LIN {X 0,Y 153.521,Z 523.718,A -85,B 0,C 180,E1 -23960.081,E2 -23960.081} C_VEL
LIN {X 0,Y 151.125,Z 510.32,A -85,B 0,C 180,E1 -23962.603,E2 -23962.603} C_VEL
LIN {X 0,Y 149.17,Z 497.902,A -85,B 0,C 180,E1 -23964.528,E2 -23964.528} C_VEL
LIN {X 0,Y 149.562,Z 497.851,A -85,B 0,C 180,E1 -23971.125,E2 -23971.125} C_VEL
LIN {X 0,Y 149.777,Z 497.824,A -85,B 0,C 180,E1 -23974.27,E2 -23974.27} C_VEL
LIN {X 0,Y 149.994,Z 497.8,A -85,B 0,C 180,E1 -23977.527,E2 -23977.527} C_VEL
LIN {X 0,Y 150.1,Z 497.781,A -85,B 0,C 180,E1 -23981.482,E2 -23981.482} C_VEL
LIN {X 0,Y 150.129,Z 497.783,A -85,B 0,C 180,E1 -23985.396,E2 -23985.396} C_VEL
LIN {X 0,Y 150.159,Z 497.776,A -85,B 0,C 180,E1 -23989.06,E2 -23989.06} C_VEL
LIN {X 0,Y 150.219,Z 497.772,A -85,B 0,C 180,E1 -23992.689,E2 -23992.689} C_VEL
LIN {X 0,Y 150.222,Z 497.77,A -85,B 0,C 180,E1 -23997.365,E2 -23997.365} C_VEL
LIN {X 0,Y 150.249,Z 497.769,A -85,B 0,C 180,E1 -24002.717,E2 -24002.717} C_VEL
LIN {X 0,Y 150.355,Z 497.751,A -85,B 0,C 180,E1 -24009.207,E2 -24009.207} C_VEL
LIN {X 0,Y 150.367,Z 497.755,A -85,B 0,C 180,E1 -24013.713,E2 -24013.713} C_VEL
LIN {X 0,Y 150.616,Z 497.721,A -85,B 0,C 180,E1 -24019.242,E2 -24019.242} C_VEL
LIN {X 0,Y 150.709,Z 497.713,A -85,B 0,C 180,E1 -24021.957,E2 -24021.957} C_VEL
LIN {X 0,Y 151.222,Z 497.65,A -85,B 0,C 180,E1 -24029.999,E2 -24029.999} C_VEL
LIN {X 0,Y 150.706,Z 497.714,A -85,B 0,C 180,E1 -24038.042,E2 -24038.042} C_VEL
LIN {X 0,Y 150.581,Z 497.726,A -85,B 0,C 180,E1 -24041.437,E2 -24041.437} C_VEL
LIN {X 0,Y 150.366,Z 497.755,A -85,B 0,C 180,E1 -24046.286,E2 -24046.286} C_VEL
LIN {X 0,Y 150.354,Z 497.751,A -85,B 0,C 180,E1 -24050.792,E2 -24050.792} C_VEL
LIN {X 0,Y 150.247,Z 497.769,A -85,B 0,C 180,E1 -24057.282,E2 -24057.282} C_VEL
LIN {X 0,Y 150.221,Z 497.77,A -85,B 0,C 180,E1 -24062.634,E2 -24062.634} C_VEL
LIN {X 0,Y 150.213,Z 497.773,A -85,B 0,C 180,E1 -24067.461,E2 -24067.461} C_VEL
LIN {X 0,Y 150.155,Z 497.778,A -85,B 0,C 180,E1 -24071.505,E2 -24071.505} C_VEL
LIN {X 0,Y 150.127,Z 497.784,A -85,B 0,C 180,E1 -24075.395,E2 -24075.395} C_VEL
LIN {X 0,Y 150.151,Z 497.775,A -85,B 0,C 180,E1 -24079.057,E2 -24079.057} C_VEL
LIN {X 0,Y 150.18,Z 497.777,A -85,B 0,C 180,E1 -24082.707,E2 -24082.707} C_VEL
LIN {X 0,Y 150.216,Z 497.767,A -85,B 0,C 180,E1 -24087.367,E2 -24087.367} C_VEL
LIN {X 0,Y 150.246,Z 497.768,A -85,B 0,C 180,E1 -24092.717,E2 -24092.717} C_VEL
LIN {X 0,Y 150.352,Z 497.756,A -85,B 0,C 180,E1 -24099.207,E2 -24099.207} C_VEL
LIN {X 0,Y 150.369,Z 497.749,A -85,B 0,C 180,E1 -24103.713,E2 -24103.713} C_VEL
LIN {X 0,Y 150.689,Z 497.715,A -85,B 0,C 180,E1 -24109.247,E2 -24109.247} C_VEL
LIN {X 0,Y 150.764,Z 497.701,A -85,B 0,C 180,E1 -24111.96,E2 -24111.96} C_VEL
LIN {X 0,Y 151.219,Z 497.646,A -85,B 0,C 180,E1 -24119.999,E2 -24119.999} C_VEL
LIN {X 0,Y 150.763,Z 497.704,A -85,B 0,C 180,E1 -24128.038,E2 -24128.038} C_VEL
LIN {X 0,Y 150.635,Z 497.716,A -85,B 0,C 180,E1 -24131.546,E2 -24131.546} C_VEL
LIN {X 0,Y 150.39,Z 497.75,A -85,B 0,C 180,E1 -24136.283,E2 -24136.283} C_VEL
LIN {X 0,Y 150.352,Z 497.751,A -85,B 0,C 180,E1 -24140.793,E2 -24140.793} C_VEL
LIN {X 0,Y 150.243,Z 497.766,A -85,B 0,C 180,E1 -24147.282,E2 -24147.282} C_VEL
LIN {X 0,Y 150.217,Z 497.772,A -85,B 0,C 180,E1 -24152.634,E2 -24152.634} C_VEL
LIN {X 0,Y 150.272,Z 497.761,A -85,B 0,C 180,E1 -24157.444,E2 -24157.444} C_VEL
LIN {X 0,Y 150.66,Z 497.722,A -85,B 0,C 180,E1 -24164.404,E2 -24164.404} C_VEL
LIN {X 0,Y 150.926,Z 497.779,A -85,B 0,C 180,E1 -24167.801,E2 -24167.801} C_VEL
LIN {X 0,Y 151.492,Z 501.356,A -85,B 0,C 180,E1 -24172.909,E2 -24172.909} C_VEL
LIN {X 0,Y 150.914,Z 503.56,A -85,B 0,C 180,E1 -24176.025,E2 -24176.025} C_VEL
LIN {X 0,Y 149.311,Z 508.708,A -85,B 0,C 180,E1 -24183.421,E2 -24183.421} C_VEL
LIN {X 0,Y 149.153,Z 509.709,A -85,B 0,C 180,E1 -24184.554,E2 -24184.554} C_VEL
LIN {X 0,Y 149.244,Z 521.963,A -85,B 0,C 180,E1 -24186.221,E2 -24186.221} C_VEL
LIN {X 0,Y 150.04,Z 534.433,A -85,B 0,C 180,E1 -24188.353,E2 -24188.353} C_VEL
LIN {X 0,Y 151.472,Z 548.682,A -85,B 0,C 180,E1 -24191.399,E2 -24191.399} C_VEL
LIN {X 0,Y 152.465,Z 556.019,A -85,B 0,C 180,E1 -24193.256,E2 -24193.256} C_VEL
LIN {X 0,Y 151.39,Z 566.543,A -85,B 0,C 180,E1 -24196.579,E2 -24196.579} C_VEL
LIN {X 0,Y 150.754,Z 575.217,A -85,B 0,C 180,E1 -24199.935,E2 -24199.935} C_VEL
LIN {X 0,Y 150.469,Z 583.731,A -85,B 0,C 180,E1 -24203.968,E2 -24203.968} C_VEL
LIN {X 0,Y 150.485,Z 590.632,A -85,B 0,C 180,E1 -24207.993,E2 -24207.993} C_VEL
LIN {X 0,Y 150.437,Z 595.255,A -85,B 0,C 180,E1 -24211.339,E2 -24211.339} C_VEL
LIN {X 0,Y 149.675,Z 599.338,A -85,B 0,C 180,E1 -24215.389,E2 -24215.389} C_VEL
LIN {X 0,Y 149.531,Z 603.504,A -85,B 0,C 180,E1 -24220.837,E2 -24220.837} C_VEL
LIN {X 0,Y 150.784,Z 606.344,A -85,B 0,C 180,E1 -24226.24,E2 -24226.24} C_VEL
LIN {X 0,Y 153.651,Z 608.104,A -85,B 0,C 180,E1 -24231.465,E2 -24231.465} C_VEL
LIN {X 0,Y 158.091,Z 608.839,A -85,B 0,C 180,E1 -24236.395,E2 -24236.395} C_VEL
LIN {X 0,Y 163.869,Z 608.541,A -85,B 0,C 180,E1 -24240.975,E2 -24240.975} C_VEL
LIN {X 0,Y 171.129,Z 607.246,A -85,B 0,C 180,E1 -24245.097,E2 -24245.097} C_VEL
LIN {X 0,Y 179.626,Z 604.926,A -85,B 0,C 180,E1 -24248.757,E2 -24248.757} C_VEL
LIN {X 0,Y 189.105,Z 601.572,A -85,B 0,C 180,E1 -24251.988,E2 -24251.988} C_VEL
LIN {X 0,Y 192.623,Z 600.091,A -85,B 0,C 180,E1 -24253.138,E2 -24253.138} C_VEL
LIN {X 0,Y 193.61,Z 599.628,A -85,B 0,C 180,E1 -24253.607,E2 -24253.607} C_VEL
LIN {X 0,Y 196.664,Z 597.909,A -85,B 0,C 180,E1 -24255.621,E2 -24255.621} C_VEL
LIN {X 0,Y 197.814,Z 597.023,A -85,B 0,C 180,E1 -24257.543,E2 -24257.543} C_VEL
LIN {X 0,Y 197.818,Z 596.879,A -85,B 0,C 180,E1 -24258.253,E2 -24258.253} C_VEL
LIN {X 0,Y 195.704,Z 597.395,A -85,B 0,C 180,E1 -24259.729,E2 -24259.729} C_VEL
LIN {X 0,Y 186.845,Z 599.739,A -85,B 0,C 180,E1 -24262.461,E2 -24262.461} C_VEL
LIN {X 0,Y 182.52,Z 600.628,A -85,B 0,C 180,E1 -24263.684,E2 -24263.684} C_VEL
LIN {X 0,Y 174.385,Z 601.787,A -85,B 0,C 180,E1 -24265.473,E2 -24265.473} C_VEL
LIN {X 0,Y 166.565,Z 602.246,A -85,B 0,C 180,E1 -24267.481,E2 -24267.481} C_VEL
LIN {X 0,Y 162.816,Z 602.037,A -85,B 0,C 180,E1 -24269.048,E2 -24269.048} C_VEL
LIN {X 0,Y 156.211,Z 600.761,A -85,B 0,C 180,E1 -24273.263,E2 -24273.263} C_VEL
LIN {X 0,Y 150.578,Z 598.332,A -85,B 0,C 180,E1 -24278.076,E2 -24278.076} C_VEL
LIN {X 0,Y 146.248,Z 594.729,A -85,B 0,C 180,E1 -24283.242,E2 -24283.242} C_VEL
LIN {X 0,Y 143.432,Z 589.927,A -85,B 0,C 180,E1 -24288.698,E2 -24288.698} C_VEL
LIN {X 0,Y 142.119,Z 583.755,A -85,B 0,C 180,E1 -24294.325,E2 -24294.325} C_VEL
LIN {X 0,Y 141.676,Z 576.967,A -85,B 0,C 180,E1 -24299.29,E2 -24299.29} C_VEL
LIN {X 0,Y 141.77,Z 569.83,A -85,B 0,C 180,E1 -24303.553,E2 -24303.553} C_VEL
LIN {X 0,Y 142.26,Z 561.329,A -85,B 0,C 180,E1 -24307.791,E2 -24307.791} C_VEL
LIN {X 0,Y 143.209,Z 550.91,A -85,B 0,C 180,E1 -24312.039,E2 -24312.039} C_VEL
LIN {X 0,Y 144.511,Z 539.254,A -85,B 0,C 180,E1 -24315.877,E2 -24315.877} C_VEL
LIN {X 0,Y 146.135,Z 526.358,A -85,B 0,C 180,E1 -24319.308,E2 -24319.308} C_VEL
LIN {X 0,Y 146.371,Z 523.299,A -85,B 0,C 180,E1 -24319.997,E2 -24319.997} C_VEL
LIN {X 0,Y 144.062,Z 510.827,A -85,B 0,C 180,E1 -24322.434,E2 -24322.434} C_VEL
LIN {X 0,Y 142.132,Z 498.779,A -85,B 0,C 180,E1 -24324.368,E2 -24324.368} C_VEL
LIN {X 0,Y 142.327,Z 498.755,A -85,B 0,C 180,E1 -24329.591,E2 -24329.591} C_VEL
LIN {X 0,Y 142.661,Z 498.708,A -85,B 0,C 180,E1 -24333.123,E2 -24333.123} C_VEL
LIN {X 0,Y 142.93,Z 498.682,A -85,B 0,C 180,E1 -24338.117,E2 -24338.117} C_VEL
LIN {X 0,Y 143.026,Z 498.665,A -85,B 0,C 180,E1 -24343.468,E2 -24343.468} C_VEL
LIN {X 0,Y 143.071,Z 498.662,A -85,B 0,C 180,E1 -24347.464,E2 -24347.464} C_VEL
LIN {X 0,Y 143.11,Z 498.654,A -85,B 0,C 180,E1 -24351.791,E2 -24351.791} C_VEL
LIN {X 0,Y 143.19,Z 498.646,A -85,B 0,C 180,E1 -24357.322,E2 -24357.322} C_VEL
LIN {X 0,Y 143.195,Z 498.647,A -85,B 0,C 180,E1 -24362.062,E2 -24362.062} C_VEL
LIN {X 0,Y 143.281,Z 498.633,A -85,B 0,C 180,E1 -24368.745,E2 -24368.745} C_VEL
LIN {X 0,Y 143.306,Z 498.633,A -85,B 0,C 180,E1 -24372.887,E2 -24372.887} C_VEL
LIN {X 0,Y 143.542,Z 498.603,A -85,B 0,C 180,E1 -24378.705,E2 -24378.705} C_VEL
LIN {X 0,Y 143.631,Z 498.594,A -85,B 0,C 180,E1 -24381.558,E2 -24381.558} C_VEL
LIN {X 0,Y 144.18,Z 498.527,A -85,B 0,C 180,E1 -24389.999,E2 -24389.999} C_VEL
LIN {X 0,Y 143.628,Z 498.594,A -85,B 0,C 180,E1 -24398.441,E2 -24398.441} C_VEL
LIN {X 0,Y 143.509,Z 498.606,A -85,B 0,C 180,E1 -24401.63,E2 -24401.63} C_VEL
LIN {X 0,Y 143.305,Z 498.633,A -85,B 0,C 180,E1 -24407.112,E2 -24407.112} C_VEL
LIN {X 0,Y 143.28,Z 498.633,A -85,B 0,C 180,E1 -24411.254,E2 -24411.254} C_VEL
LIN {X 0,Y 143.193,Z 498.647,A -85,B 0,C 180,E1 -24417.937,E2 -24417.937} C_VEL
LIN {X 0,Y 143.171,Z 498.649,A -85,B 0,C 180,E1 -24423.435,E2 -24423.435} C_VEL
LIN {X 0,Y 143.076,Z 498.657,A -85,B 0,C 180,E1 -24429.684,E2 -24429.684} C_VEL
LIN {X 0,Y 143.058,Z 498.665,A -85,B 0,C 180,E1 -24433.454,E2 -24433.454} C_VEL
LIN {X 0,Y 143.066,Z 498.659,A -85,B 0,C 180,E1 -24437.464,E2 -24437.464} C_VEL
LIN {X 0,Y 143.079,Z 498.663,A -85,B 0,C 180,E1 -24441.805,E2 -24441.805} C_VEL
LIN {X 0,Y 143.183,Z 498.643,A -85,B 0,C 180,E1 -24447.321,E2 -24447.321} C_VEL
LIN {X 0,Y 143.192,Z 498.648,A -85,B 0,C 180,E1 -24452.061,E2 -24452.061} C_VEL
LIN {X 0,Y 143.278,Z 498.636,A -85,B 0,C 180,E1 -24458.744,E2 -24458.744} C_VEL
LIN {X 0,Y 143.306,Z 498.631,A -85,B 0,C 180,E1 -24462.887,E2 -24462.887} C_VEL
LIN {X 0,Y 143.603,Z 498.596,A -85,B 0,C 180,E1 -24468.71,E2 -24468.71} C_VEL
LIN {X 0,Y 143.685,Z 498.584,A -85,B 0,C 180,E1 -24471.561,E2 -24471.561} C_VEL
LIN {X 0,Y 144.178,Z 498.523,A -85,B 0,C 180,E1 -24479.999,E2 -24479.999} C_VEL
LIN {X 0,Y 143.685,Z 498.585,A -85,B 0,C 180,E1 -24488.437,E2 -24488.437} C_VEL
LIN {X 0,Y 143.571,Z 498.597,A -85,B 0,C 180,E1 -24491.757,E2 -24491.757} C_VEL
LIN {X 0,Y 143.323,Z 498.632,A -85,B 0,C 180,E1 -24497.11,E2 -24497.11} C_VEL
LIN {X 0,Y 143.277,Z 498.634,A -85,B 0,C 180,E1 -24501.255,E2 -24501.255} C_VEL
LIN {X 0,Y 143.189,Z 498.642,A -85,B 0,C 180,E1 -24507.937,E2 -24507.937} C_VEL
LIN {X 0,Y 143.169,Z 498.652,A -85,B 0,C 180,E1 -24513.436,E2 -24513.436} C_VEL
LIN {X 0,Y 143.235,Z 498.642,A -85,B 0,C 180,E1 -24519.632,E2 -24519.632} C_VEL
LIN {X 0,Y 143.47,Z 498.614,A -85,B 0,C 180,E1 -24523.298,E2 -24523.298} C_VEL
LIN {X 0,Y 143.966,Z 498.62,A -85,B 0,C 180,E1 -24528.703,E2 -24528.703} C_VEL
LIN {X 0,Y 144.404,Z 501.33,A -85,B 0,C 180,E1 -24532.773,E2 -24532.773} C_VEL
LIN {X 0,Y 143.396,Z 504.406,A -85,B 0,C 180,E1 -24537.377,E2 -24537.377} C_VEL
LIN {X 0,Y 142.08,Z 509.031,A -85,B 0,C 180,E1 -24544.452,E2 -24544.452} C_VEL
LIN {X 0,Y 142.227,Z 522.949,A -85,B 0,C 180,E1 -24546.522,E2 -24546.522} C_VEL
LIN {X 0,Y 143.214,Z 536.813,A -85,B 0,C 180,E1 -24549.131,E2 -24549.131} C_VEL
LIN {X 0,Y 144.534,Z 549.001,A -85,B 0,C 180,E1 -24551.942,E2 -24551.942} C_VEL
LIN {X 0,Y 145.421,Z 554.89,A -85,B 0,C 180,E1 -24553.506,E2 -24553.506} C_VEL
LIN {X 0,Y 144.47,Z 565.324,A -85,B 0,C 180,E1 -24556.981,E2 -24556.981} C_VEL
LIN {X 0,Y 143.853,Z 574.877,A -85,B 0,C 180,E1 -24560.864,E2 -24560.864} C_VEL
LIN {X 0,Y 143.686,Z 583.335,A -85,B 0,C 180,E1 -24565.09,E2 -24565.09} C_VEL
LIN {X 0,Y 143.719,Z 589.07,A -85,B 0,C 180,E1 -24568.6,E2 -24568.6} C_VEL
LIN {X 0,Y 143.714,Z 592.828,A -85,B 0,C 180,E1 -24571.402,E2 -24571.402} C_VEL
LIN {X 0,Y 143.198,Z 595.868,A -85,B 0,C 180,E1 -24574.222,E2 -24574.222} C_VEL
LIN {X 0,Y 142.722,Z 600.711,A -85,B 0,C 180,E1 -24579.988,E2 -24579.988} C_VEL
LIN {X 0,Y 143.292,Z 603.359,A -85,B 0,C 180,E1 -24584.196,E2 -24584.196} C_VEL
LIN {X 0,Y 145.395,Z 605.94,A -85,B 0,C 180,E1 -24589.778,E2 -24589.778} C_VEL
LIN {X 0,Y 149.33,Z 607.531,A -85,B 0,C 180,E1 -24595.061,E2 -24595.061} C_VEL
LIN {X 0,Y 154.681,Z 608.094,A -85,B 0,C 180,E1 -24599.987,E2 -24599.987} C_VEL
LIN {X 0,Y 161.446,Z 607.693,A -85,B 0,C 180,E1 -24604.466,E2 -24604.466} C_VEL
LIN {X 0,Y 169.632,Z 606.322,A -85,B 0,C 180,E1 -24608.424,E2 -24608.424} C_VEL
LIN {X 0,Y 178.912,Z 603.955,A -85,B 0,C 180,E1 -24611.898,E2 -24611.898} C_VEL
LIN {X 0,Y 183.913,Z 602.406,A -85,B 0,C 180,E1 -24613.461,E2 -24613.461} C_VEL
LIN {X 0,Y 188.351,Z 600.741,A -85,B 0,C 180,E1 -24615.15,E2 -24615.15} C_VEL
LIN {X 0,Y 190.86,Z 599.403,A -85,B 0,C 180,E1 -24617.431,E2 -24617.431} C_VEL
LIN {X 0,Y 190.34,Z 599.38,A -85,B 0,C 180,E1 -24618.347,E2 -24618.347} C_VEL
LIN {X 0,Y 180.398,Z 601.373,A -85,B 0,C 180,E1 -24621.441,E2 -24621.441} C_VEL
LIN {X 0,Y 171.242,Z 602.278,A -85,B 0,C 180,E1 -24624.93,E2 -24624.93} C_VEL
LIN {X 0,Y 162.816,Z 602.037,A -85,B 0,C 180,E1 -24629.048,E2 -24629.048} C_VEL
LIN {X 0,Y 159.227,Z 601.639,A -85,B 0,C 180,E1 -24630.708,E2 -24630.708} C_VEL
LIN {X 0,Y 152.249,Z 600.466,A -85,B 0,C 180,E1 -24633.261,E2 -24633.261} C_VEL
LIN {X 0,Y 145.778,Z 598.59,A -85,B 0,C 180,E1 -24636.045,E2 -24636.045} C_VEL
LIN {X 0,Y 143.074,Z 597.163,A -85,B 0,C 180,E1 -24638.044,E2 -24638.044} C_VEL
LIN {X 0,Y 138.628,Z 592.71,A -85,B 0,C 180,E1 -24643.81,E2 -24643.81} C_VEL
LIN {X 0,Y 136.116,Z 587.195,A -85,B 0,C 180,E1 -24649.635,E2 -24649.635} C_VEL
LIN {X 0,Y 135.22,Z 582.148,A -85,B 0,C 180,E1 -24654.034,E2 -24654.034} C_VEL
LIN {X 0,Y 134.779,Z 574.999,A -85,B 0,C 180,E1 -24659.254,E2 -24659.254} C_VEL
LIN {X 0,Y 134.894,Z 567.52,A -85,B 0,C 180,E1 -24663.735,E2 -24663.735} C_VEL
LIN {X 0,Y 135.401,Z 558.506,A -85,B 0,C 180,E1 -24668.188,E2 -24668.188} C_VEL
LIN {X 0,Y 136.447,Z 547.54,A -85,B 0,C 180,E1 -24672.646,E2 -24672.646} C_VEL
LIN {X 0,Y 137.713,Z 536.486,A -85,B 0,C 180,E1 -24676.302,E2 -24676.302} C_VEL
LIN {X 0,Y 139.214,Z 524.261,A -85,B 0,C 180,E1 -24679.54,E2 -24679.54} C_VEL
LIN {X 0,Y 138.497,Z 519.379,A -85,B 0,C 180,E1 -24680.613,E2 -24680.613} C_VEL
LIN {X 0,Y 136.138,Z 506.12,A -85,B 0,C 180,E1 -24683.145,E2 -24683.145} C_VEL
LIN {X 0,Y 135.091,Z 499.655,A -85,B 0,C 180,E1 -24684.279,E2 -24684.279} C_VEL
LIN {X 0,Y 135.394,Z 499.616,A -85,B 0,C 180,E1 -24691.271,E2 -24691.271} C_VEL
LIN {X 0,Y 135.681,Z 499.582,A -85,B 0,C 180,E1 -24694.736,E2 -24694.736} C_VEL
LIN {X 0,Y 135.927,Z 499.551,A -85,B 0,C 180,E1 -24699.143,E2 -24699.143} C_VEL
LIN {X 0,Y 135.973,Z 499.544,A -85,B 0,C 180,E1 -24703.645,E2 -24703.645} C_VEL
LIN {X 0,Y 136.035,Z 499.539,A -85,B 0,C 180,E1 -24707.807,E2 -24707.807} C_VEL
LIN {X 0,Y 136.059,Z 499.531,A -85,B 0,C 180,E1 -24711.694,E2 -24711.694} C_VEL
LIN {X 0,Y 136.094,Z 499.532,A -85,B 0,C 180,E1 -24715.717,E2 -24715.717} C_VEL
LIN {X 0,Y 136.151,Z 499.526,A -85,B 0,C 180,E1 -24722.317,E2 -24722.317} C_VEL
LIN {X 0,Y 136.248,Z 499.509,A -85,B 0,C 180,E1 -24728.833,E2 -24728.833} C_VEL
LIN {X 0,Y 136.273,Z 499.507,A -85,B 0,C 180,E1 -24735.056,E2 -24735.056} C_VEL
LIN {X 0,Y 136.449,Z 499.484,A -85,B 0,C 180,E1 -24738.138,E2 -24738.138} C_VEL
LIN {X 0,Y 136.556,Z 499.474,A -85,B 0,C 180,E1 -24741.117,E2 -24741.117} C_VEL
LIN {X 0,Y 137.137,Z 499.404,A -85,B 0,C 180,E1 -24749.999,E2 -24749.999} C_VEL
LIN {X 0,Y 136.553,Z 499.474,A -85,B 0,C 180,E1 -24758.881,E2 -24758.881} C_VEL
LIN {X 0,Y 136.444,Z 499.484,A -85,B 0,C 180,E1 -24761.889,E2 -24761.889} C_VEL
LIN {X 0,Y 136.245,Z 499.514,A -85,B 0,C 180,E1 -24768.028,E2 -24768.028} C_VEL
LIN {X 0,Y 136.201,Z 499.513,A -85,B 0,C 180,E1 -24771.748,E2 -24771.748} C_VEL
LIN {X 0,Y 136.103,Z 499.528,A -85,B 0,C 180,E1 -24778.616,E2 -24778.616} C_VEL
LIN {X 0,Y 136.081,Z 499.533,A -85,B 0,C 180,E1 -24784.617,E2 -24784.617} C_VEL
LIN {X 0,Y 136.052,Z 499.532,A -85,B 0,C 180,E1 -24789.207,E2 -24789.207} C_VEL
LIN {X 0,Y 136,Z 499.545,A -85,B 0,C 180,E1 -24793.657,E2 -24793.657} C_VEL
LIN {X 0,Y 136.006,Z 499.537,A -85,B 0,C 180,E1 -24797.795,E2 -24797.795} C_VEL
LIN {X 0,Y 136.028,Z 499.541,A -85,B 0,C 180,E1 -24801.683,E2 -24801.683} C_VEL
LIN {X 0,Y 136.056,Z 499.533,A -85,B 0,C 180,E1 -24805.738,E2 -24805.738} C_VEL
LIN {X 0,Y 136.148,Z 499.525,A -85,B 0,C 180,E1 -24812.316,E2 -24812.316} C_VEL
LIN {X 0,Y 136.245,Z 499.512,A -85,B 0,C 180,E1 -24818.832,E2 -24818.832} C_VEL
LIN {X 0,Y 136.278,Z 499.502,A -85,B 0,C 180,E1 -24825.056,E2 -24825.056} C_VEL
LIN {X 0,Y 136.501,Z 499.481,A -85,B 0,C 180,E1 -24828.114,E2 -24828.114} C_VEL
LIN {X 0,Y 136.609,Z 499.467,A -85,B 0,C 180,E1 -24831.121,E2 -24831.121} C_VEL
LIN {X 0,Y 137.135,Z 499.4,A -85,B 0,C 180,E1 -24839.999,E2 -24839.999} C_VEL
LIN {X 0,Y 136.609,Z 499.467,A -85,B 0,C 180,E1 -24848.878,E2 -24848.878} C_VEL
LIN {X 0,Y 136.493,Z 499.479,A -85,B 0,C 180,E1 -24851.958,E2 -24851.958} C_VEL
LIN {X 0,Y 136.257,Z 499.508,A -85,B 0,C 180,E1 -24858.027,E2 -24858.027} C_VEL
LIN {X 0,Y 136.198,Z 499.518,A -85,B 0,C 180,E1 -24861.75,E2 -24861.75} C_VEL
LIN {X 0,Y 136.099,Z 499.524,A -85,B 0,C 180,E1 -24868.616,E2 -24868.616} C_VEL
LIN {X 0,Y 136.088,Z 499.532,A -85,B 0,C 180,E1 -24874.616,E2 -24874.616} C_VEL
LIN {X 0,Y 136.179,Z 499.519,A -85,B 0,C 180,E1 -24879.275,E2 -24879.275} C_VEL
LIN {X 0,Y 136.637,Z 499.464,A -85,B 0,C 180,E1 -24886.062,E2 -24886.062} C_VEL
LIN {X 0,Y 136.997,Z 499.543,A -85,B 0,C 180,E1 -24889.896,E2 -24889.896} C_VEL
LIN {X 0,Y 137.229,Z 500.924,A -85,B 0,C 180,E1 -24892.081,E2 -24892.081} C_VEL
LIN {X 0,Y 136.801,Z 502.939,A -85,B 0,C 180,E1 -24895.283,E2 -24895.283} C_VEL
LIN {X 0,Y 135.342,Z 507.194,A -85,B 0,C 180,E1 -24902.138,E2 -24902.138} C_VEL
LIN {X 0,Y 135.005,Z 508.681,A -85,B 0,C 180,E1 -24904.567,E2 -24904.567} C_VEL
LIN {X 0,Y 135.085,Z 521.4,A -85,B 0,C 180,E1 -24906.527,E2 -24906.527} C_VEL
LIN {X 0,Y 136.027,Z 535.132,A -85,B 0,C 180,E1 -24909.195,E2 -24909.195} C_VEL
LIN {X 0,Y 137.384,Z 547.414,A -85,B 0,C 180,E1 -24912.126,E2 -24912.126} C_VEL
LIN {X 0,Y 138.4,Z 554.001,A -85,B 0,C 180,E1 -24913.934,E2 -24913.934} C_VEL
LIN {X 0,Y 137.59,Z 564.073,A -85,B 0,C 180,E1 -24917.429,E2 -24917.429} C_VEL
LIN {X 0,Y 137.047,Z 572.946,A -85,B 0,C 180,E1 -24921.151,E2 -24921.151} C_VEL
LIN {X 0,Y 136.934,Z 581.541,A -85,B 0,C 180,E1 -24925.585,E2 -24925.585} C_VEL
LIN {X 0,Y 137.016,Z 588.378,A -85,B 0,C 180,E1 -24930.001,E2 -24930.001} C_VEL
LIN {X 0,Y 136.852,Z 592.022,A -85,B 0,C 180,E1 -24932.944,E2 -24932.944} C_VEL
LIN {X 0,Y 136.035,Z 597.452,A -85,B 0,C 180,E1 -24938.917,E2 -24938.917} C_VEL
LIN {X 0,Y 136.631,Z 601.525,A -85,B 0,C 180,E1 -24944.904,E2 -24944.904} C_VEL
LIN {X 0,Y 138.872,Z 604.406,A -85,B 0,C 180,E1 -24950.749,E2 -24950.749} C_VEL
LIN {X 0,Y 143.002,Z 606.304,A -85,B 0,C 180,E1 -24956.253,E2 -24956.253} C_VEL
LIN {X 0,Y 148.6,Z 607.22,A -85,B 0,C 180,E1 -24961.349,E2 -24961.349} C_VEL
LIN {X 0,Y 155.663,Z 607.204,A -85,B 0,C 180,E1 -24965.941,E2 -24965.941} C_VEL
LIN {X 0,Y 164.135,Z 606.26,A -85,B 0,C 180,E1 -24969.963,E2 -24969.963} C_VEL
LIN {X 0,Y 173.706,Z 604.359,A -85,B 0,C 180,E1 -24973.457,E2 -24973.457} C_VEL
LIN {X 0,Y 178.839,Z 603.047,A -85,B 0,C 180,E1 -24975.021,E2 -24975.021} C_VEL
LIN {X 0,Y 182.913,Z 601.688,A -85,B 0,C 180,E1 -24976.89,E2 -24976.89} C_VEL
LIN {X 0,Y 180.034,Z 601.984,A -85,B 0,C 180,E1 -24978.423,E2 -24978.423} C_VEL
LIN {X 0,Y 169.911,Z 602.975,A -85,B 0,C 180,E1 -24981.804,E2 -24981.804} C_VEL
LIN {X 0,Y 161.223,Z 602.863,A -85,B 0,C 180,E1 -24985.48,E2 -24985.48} C_VEL
LIN {X 0,Y 153.324,Z 601.682,A -85,B 0,C 180,E1 -24989.721,E2 -24989.721} C_VEL
LIN {X 0,Y 146.749,Z 599.415,A -85,B 0,C 180,E1 -24994.468,E2 -24994.468} C_VEL
LIN {X 0,Y 143.074,Z 597.163,A -85,B 0,C 180,E1 -24998.044,E2 -24998.044} C_VEL
LIN {X 0,Y 140.599,Z 595.583,A -85,B 0,C 180,E1 -25000.104,E2 -25000.104} C_VEL
LIN {X 0,Y 135.387,Z 592.295,A -85,B 0,C 180,E1 -25003.322,E2 -25003.322} C_VEL
LIN {X 0,Y 130.782,Z 588.321,A -85,B 0,C 180,E1 -25006.709,E2 -25006.709} C_VEL
LIN {X 0,Y 129.343,Z 585.771,A -85,B 0,C 180,E1 -25008.979,E2 -25008.979} C_VEL
LIN {X 0,Y 128.353,Z 580.408,A -85,B 0,C 180,E1 -25013.714,E2 -25013.714} C_VEL
LIN {X 0,Y 127.958,Z 572.813,A -85,B 0,C 180,E1 -25019.214,E2 -25019.214} C_VEL
LIN {X 0,Y 128.057,Z 564.956,A -85,B 0,C 180,E1 -25023.934,E2 -25023.934} C_VEL
LIN {X 0,Y 128.537,Z 556.37,A -85,B 0,C 180,E1 -25028.219,E2 -25028.219} C_VEL
LIN {X 0,Y 129.525,Z 545.913,A -85,B 0,C 180,E1 -25032.536,E2 -25032.536} C_VEL
LIN {X 0,Y 130.95,Z 533.271,A -85,B 0,C 180,E1 -25036.767,E2 -25036.767} C_VEL
LIN {X 0,Y 132.118,Z 523.607,A -85,B 0,C 180,E1 -25039.42,E2 -25039.42} C_VEL
LIN {X 0,Y 129.791,Z 511.029,A -85,B 0,C 180,E1 -25042.1,E2 -25042.1} C_VEL
LIN {X 0,Y 128.1,Z 500.525,A -85,B 0,C 180,E1 -25043.974,E2 -25043.974} C_VEL
LIN {X 0,Y 128.179,Z 500.518,A -85,B 0,C 180,E1 -25049.57,E2 -25049.57} C_VEL
LIN {X 0,Y 128.634,Z 500.46,A -85,B 0,C 180,E1 -25054.96,E2 -25054.96} C_VEL
LIN {X 0,Y 128.855,Z 500.428,A -85,B 0,C 180,E1 -25060.883,E2 -25060.883} C_VEL
LIN {X 0,Y 128.919,Z 500.425,A -85,B 0,C 180,E1 -25065.13,E2 -25065.13} C_VEL
LIN {X 0,Y 128.961,Z 500.416,A -85,B 0,C 180,E1 -25069.728,E2 -25069.728} C_VEL
LIN {X 0,Y 128.996,Z 500.416,A -85,B 0,C 180,E1 -25074.811,E2 -25074.811} C_VEL
LIN {X 0,Y 129.037,Z 500.408,A -85,B 0,C 180,E1 -25080.646,E2 -25080.646} C_VEL
LIN {X 0,Y 129.112,Z 500.396,A -85,B 0,C 180,E1 -25087.602,E2 -25087.602} C_VEL
LIN {X 0,Y 129.158,Z 500.395,A -85,B 0,C 180,E1 -25090.944,E2 -25090.944} C_VEL
LIN {X 0,Y 129.37,Z 500.364,A -85,B 0,C 180,E1 -25097.922,E2 -25097.922} C_VEL
LIN {X 0,Y 129.481,Z 500.356,A -85,B 0,C 180,E1 -25100.628,E2 -25100.628} C_VEL
LIN {X 0,Y 130.092,Z 500.281,A -85,B 0,C 180,E1 -25109.999,E2 -25109.999} C_VEL
LIN {X 0,Y 129.479,Z 500.356,A -85,B 0,C 180,E1 -25119.371,E2 -25119.371} C_VEL
LIN {X 0,Y 129.347,Z 500.366,A -85,B 0,C 180,E1 -25122.552,E2 -25122.552} C_VEL
LIN {X 0,Y 129.157,Z 500.395,A -85,B 0,C 180,E1 -25129.055,E2 -25129.055} C_VEL
LIN {X 0,Y 129.111,Z 500.396,A -85,B 0,C 180,E1 -25132.397,E2 -25132.397} C_VEL
LIN {X 0,Y 129.038,Z 500.408,A -85,B 0,C 180,E1 -25139.372,E2 -25139.372} C_VEL
LIN {X 0,Y 128.994,Z 500.416,A -85,B 0,C 180,E1 -25145.188,E2 -25145.188} C_VEL
LIN {X 0,Y 128.952,Z 500.418,A -85,B 0,C 180,E1 -25150.844,E2 -25150.844} C_VEL
LIN {X 0,Y 128.923,Z 500.425,A -85,B 0,C 180,E1 -25155.126,E2 -25155.126} C_VEL
LIN {X 0,Y 128.943,Z 500.419,A -85,B 0,C 180,E1 -25159.734,E2 -25159.734} C_VEL
LIN {X 0,Y 128.96,Z 500.419,A -85,B 0,C 180,E1 -25164.831,E2 -25164.831} C_VEL
LIN {X 0,Y 129.052,Z 500.409,A -85,B 0,C 180,E1 -25170.65,E2 -25170.65} C_VEL
LIN {X 0,Y 129.108,Z 500.4,A -85,B 0,C 180,E1 -25177.727,E2 -25177.727} C_VEL
LIN {X 0,Y 129.156,Z 500.396,A -85,B 0,C 180,E1 -25180.943,E2 -25180.943} C_VEL
LIN {X 0,Y 129.418,Z 500.365,A -85,B 0,C 180,E1 -25187.815,E2 -25187.815} C_VEL
LIN {X 0,Y 129.531,Z 500.348,A -85,B 0,C 180,E1 -25190.631,E2 -25190.631} C_VEL
LIN {X 0,Y 130.09,Z 500.277,A -85,B 0,C 180,E1 -25199.999,E2 -25199.999} C_VEL
LIN {X 0,Y 129.531,Z 500.346,A -85,B 0,C 180,E1 -25209.367,E2 -25209.367} C_VEL
LIN {X 0,Y 129.395,Z 500.363,A -85,B 0,C 180,E1 -25212.547,E2 -25212.547} C_VEL
LIN {X 0,Y 129.163,Z 500.39,A -85,B 0,C 180,E1 -25219.054,E2 -25219.054} C_VEL
LIN {X 0,Y 129.108,Z 500.401,A -85,B 0,C 180,E1 -25222.398,E2 -25222.398} C_VEL
LIN {X 0,Y 129.035,Z 500.406,A -85,B 0,C 180,E1 -25229.373,E2 -25229.373} C_VEL
LIN {X 0,Y 129.036,Z 500.409,A -85,B 0,C 180,E1 -25235.217,E2 -25235.217} C_VEL
LIN {X 0,Y 129.174,Z 500.393,A -85,B 0,C 180,E1 -25240.759,E2 -25240.759} C_VEL
LIN {X 0,Y 129.485,Z 500.357,A -85,B 0,C 180,E1 -25245.123,E2 -25245.123} C_VEL
LIN {X 0,Y 130.011,Z 500.292,A -85,B 0,C 180,E1 -25250.943,E2 -25250.943} C_VEL
LIN {X 0,Y 129.902,Z 502.235,A -85,B 0,C 180,E1 -25254.246,E2 -25254.246} C_VEL
LIN {X 0,Y 128.391,Z 506.267,A -85,B 0,C 180,E1 -25261.142,E2 -25261.142} C_VEL
LIN {X 0,Y 127.932,Z 508.442,A -85,B 0,C 180,E1 -25264.694,E2 -25264.694} C_VEL
LIN {X 0,Y 128.014,Z 521.116,A -85,B 0,C 180,E1 -25266.76,E2 -25266.76} C_VEL
LIN {X 0,Y 128.876,Z 533.61,A -85,B 0,C 180,E1 -25269.301,E2 -25269.301} C_VEL
LIN {X 0,Y 130.453,Z 547.426,A -85,B 0,C 180,E1 -25272.766,E2 -25272.766} C_VEL
LIN {X 0,Y 131.45,Z 553.398,A -85,B 0,C 180,E1 -25274.496,E2 -25274.496} C_VEL
LIN {X 0,Y 130.632,Z 563.777,A -85,B 0,C 180,E1 -25278.361,E2 -25278.361} C_VEL
LIN {X 0,Y 130.251,Z 572.382,A -85,B 0,C 180,E1 -25282.248,E2 -25282.248} C_VEL
LIN {X 0,Y 130.285,Z 580.925,A -85,B 0,C 180,E1 -25286.908,E2 -25286.908} C_VEL
LIN {X 0,Y 130.345,Z 586.633,A -85,B 0,C 180,E1 -25290.773,E2 -25290.773} C_VEL
LIN {X 0,Y 130.225,Z 589.418,A -85,B 0,C 180,E1 -25293.094,E2 -25293.094} C_VEL
LIN {X 0,Y 129.383,Z 595.19,A -85,B 0,C 180,E1 -25299.379,E2 -25299.379} C_VEL
LIN {X 0,Y 130.032,Z 599.519,A -85,B 0,C 180,E1 -25305.679,E2 -25305.679} C_VEL
LIN {X 0,Y 132.441,Z 602.726,A -85,B 0,C 180,E1 -25311.806,E2 -25311.806} C_VEL
LIN {X 0,Y 136.765,Z 604.943,A -85,B 0,C 180,E1 -25317.548,E2 -25317.548} C_VEL
LIN {X 0,Y 144.864,Z 606.402,A -85,B 0,C 180,E1 -25324.438,E2 -25324.438} C_VEL
LIN {X 0,Y 154.247,Z 606.397,A -85,B 0,C 180,E1 -25329.635,E2 -25329.635} C_VEL
LIN {X 0,Y 163.577,Z 605.41,A -85,B 0,C 180,E1 -25333.428,E2 -25333.428} C_VEL
LIN {X 0,Y 173.822,Z 603.497,A -85,B 0,C 180,E1 -25336.701,E2 -25336.701} C_VEL
LIN {X 0,Y 169.652,Z 603.667,A -85,B 0,C 180,E1 -25338.486,E2 -25338.486} C_VEL
LIN {X 0,Y 159.905,Z 603.639,A -85,B 0,C 180,E1 -25342.026,E2 -25342.026} C_VEL
LIN {X 0,Y 151.168,Z 602.556,A -85,B 0,C 180,E1 -25346.09,E2 -25346.09} C_VEL
LIN {X 0,Y 143.713,Z 600.412,A -85,B 0,C 180,E1 -25350.724,E2 -25350.724} C_VEL
LIN {X 0,Y 137.574,Z 597.216,A -85,B 0,C 180,E1 -25355.878,E2 -25355.878} C_VEL
LIN {X 0,Y 132.852,Z 592.884,A -85,B 0,C 180,E1 -25361.494,E2 -25361.494} C_VEL
LIN {X 0,Y 129.78,Z 587.323,A -85,B 0,C 180,E1 -25367.491,E2 -25367.491} C_VEL
LIN {X 0,Y 129.343,Z 585.771,A -85,B 0,C 180,E1 -25368.979,E2 -25368.979} C_VEL
LIN {X 0,Y 128.156,Z 583.114,A -85,B 0,C 180,E1 -25371.24,E2 -25371.24} C_VEL
LIN {X 0,Y 124.877,Z 577.95,A -85,B 0,C 180,E1 -25374.747,E2 -25374.747} C_VEL
LIN {X 0,Y 122.325,Z 573.283,A -85,B 0,C 180,E1 -25377.55,E2 -25377.55} C_VEL
LIN {X 0,Y 121.246,Z 569.623,A -85,B 0,C 180,E1 -25379.742,E2 -25379.742} C_VEL
LIN {X 0,Y 121.151,Z 568.402,A -85,B 0,C 180,E1 -25380.497,E2 -25380.497} C_VEL
LIN {X 0,Y 121.469,Z 559.01,A -85,B 0,C 180,E1 -25385.812,E2 -25385.812} C_VEL
LIN {X 0,Y 122.336,Z 547.222,A -85,B 0,C 180,E1 -25391.234,E2 -25391.234} C_VEL
LIN {X 0,Y 123.661,Z 534.968,A -85,B 0,C 180,E1 -25395.662,E2 -25395.662} C_VEL
LIN {X 0,Y 124.996,Z 524.135,A -85,B 0,C 180,E1 -25398.863,E2 -25398.863} C_VEL
LIN {X 0,Y 124.043,Z 518.204,A -85,B 0,C 180,E1 -25400.284,E2 -25400.284} C_VEL
LIN {X 0,Y 121.36,Z 503.25,A -85,B 0,C 180,E1 -25403.299,E2 -25403.299} C_VEL
LIN {X 0,Y 121.077,Z 501.4,A -85,B 0,C 180,E1 -25403.689,E2 -25403.689} C_VEL
LIN {X 0,Y 121.226,Z 501.381,A -85,B 0,C 180,E1 -25411.452,E2 -25411.452} C_VEL
LIN {X 0,Y 121.621,Z 501.334,A -85,B 0,C 180,E1 -25416,E2 -25416} C_VEL
LIN {X 0,Y 121.796,Z 501.306,A -85,B 0,C 180,E1 -25421.396,E2 -25421.396} C_VEL
LIN {X 0,Y 121.847,Z 501.308,A -85,B 0,C 180,E1 -25426.199,E2 -25426.199} C_VEL
LIN {X 0,Y 121.877,Z 501.297,A -85,B 0,C 180,E1 -25430.63,E2 -25430.63} C_VEL
LIN {X 0,Y 121.949,Z 501.294,A -85,B 0,C 180,E1 -25434.808,E2 -25434.808} C_VEL
LIN {X 0,Y 121.946,Z 501.287,A -85,B 0,C 180,E1 -25439.826,E2 -25439.826} C_VEL
LIN {X 0,Y 121.987,Z 501.286,A -85,B 0,C 180,E1 -25446.215,E2 -25446.215} C_VEL
LIN {X 0,Y 122.049,Z 501.278,A -85,B 0,C 180,E1 -25449.787,E2 -25449.787} C_VEL
LIN {X 0,Y 122.243,Z 501.25,A -85,B 0,C 180,E1 -25456.704,E2 -25456.704} C_VEL
LIN {X 0,Y 122.411,Z 501.237,A -85,B 0,C 180,E1 -25460.081,E2 -25460.081} C_VEL
LIN {X 0,Y 122.603,Z 501.209,A -85,B 0,C 180,E1 -25466.713,E2 -25466.713} C_VEL
LIN {X 0,Y 123.045,Z 501.159,A -85,B 0,C 180,E1 -25469.999,E2 -25469.999} C_VEL
LIN {X 0,Y 122.426,Z 501.233,A -85,B 0,C 180,E1 -25476.592,E2 -25476.592} C_VEL
LIN {X 0,Y 122.321,Z 501.241,A -85,B 0,C 180,E1 -25482.375,E2 -25482.375} C_VEL
LIN {X 0,Y 122.112,Z 501.273,A -85,B 0,C 180,E1 -25486.724,E2 -25486.724} C_VEL
LIN {X 0,Y 122.026,Z 501.279,A -85,B 0,C 180,E1 -25492.85,E2 -25492.85} C_VEL
LIN {X 0,Y 121.952,Z 501.294,A -85,B 0,C 180,E1 -25497.453,E2 -25497.453} C_VEL
LIN {X 0,Y 121.914,Z 501.291,A -85,B 0,C 180,E1 -25501.253,E2 -25501.253} C_VEL
LIN {X 0,Y 121.914,Z 501.298,A -85,B 0,C 180,E1 -25506.188,E2 -25506.188} C_VEL
LIN {X 0,Y 121.886,Z 501.299,A -85,B 0,C 180,E1 -25511.444,E2 -25511.444} C_VEL
LIN {X 0,Y 121.873,Z 501.297,A -85,B 0,C 180,E1 -25518.56,E2 -25518.56} C_VEL
LIN {X 0,Y 121.912,Z 501.297,A -85,B 0,C 180,E1 -25524.795,E2 -25524.795} C_VEL
LIN {X 0,Y 121.94,Z 501.295,A -85,B 0,C 180,E1 -25529.827,E2 -25529.827} C_VEL
LIN {X 0,Y 121.984,Z 501.284,A -85,B 0,C 180,E1 -25536.214,E2 -25536.214} C_VEL
LIN {X 0,Y 122.047,Z 501.283,A -85,B 0,C 180,E1 -25539.786,E2 -25539.786} C_VEL
LIN {X 0,Y 122.365,Z 501.242,A -85,B 0,C 180,E1 -25547.521,E2 -25547.521} C_VEL
LIN {X 0,Y 122.457,Z 501.23,A -85,B 0,C 180,E1 -25550.085,E2 -25550.085} C_VEL
LIN {X 0,Y 122.611,Z 501.211,A -85,B 0,C 180,E1 -25556.713,E2 -25556.713} C_VEL
LIN {X 0,Y 123.044,Z 501.155,A -85,B 0,C 180,E1 -25559.999,E2 -25559.999} C_VEL
LIN {X 0,Y 122.456,Z 501.231,A -85,B 0,C 180,E1 -25566.59,E2 -25566.59} C_VEL
LIN {X 0,Y 122.457,Z 501.225,A -85,B 0,C 180,E1 -25569.914,E2 -25569.914} C_VEL
LIN {X 0,Y 122.265,Z 501.253,A -85,B 0,C 180,E1 -25573.292,E2 -25573.292} C_VEL
LIN {X 0,Y 122.051,Z 501.275,A -85,B 0,C 180,E1 -25580.211,E2 -25580.211} C_VEL
LIN {X 0,Y 121.983,Z 501.29,A -85,B 0,C 180,E1 -25583.784,E2 -25583.784} C_VEL
LIN {X 0,Y 121.941,Z 501.292,A -85,B 0,C 180,E1 -25590.174,E2 -25590.174} C_VEL
LIN {X 0,Y 122.006,Z 501.282,A -85,B 0,C 180,E1 -25596.25,E2 -25596.25} C_VEL
LIN {X 0,Y 122.287,Z 501.253,A -85,B 0,C 180,E1 -25603.602,E2 -25603.602} C_VEL
LIN {X 0,Y 122.67,Z 501.204,A -85,B 0,C 180,E1 -25608.141,E2 -25608.141} C_VEL
LIN {X 0,Y 122.951,Z 501.183,A -85,B 0,C 180,E1 -25612.546,E2 -25612.546} C_VEL
LIN {X 0,Y 122.158,Z 503.59,A -85,B 0,C 180,E1 -25616.87,E2 -25616.87} C_VEL
LIN {X 0,Y 120.865,Z 507.874,A -85,B 0,C 180,E1 -25624.837,E2 -25624.837} C_VEL
LIN {X 0,Y 121.011,Z 521.527,A -85,B 0,C 180,E1 -25627.238,E2 -25627.238} C_VEL
LIN {X 0,Y 122.033,Z 534.973,A -85,B 0,C 180,E1 -25630.225,E2 -25630.225} C_VEL
LIN {X 0,Y 123.551,Z 547.07,A -85,B 0,C 180,E1 -25633.477,E2 -25633.477} C_VEL
LIN {X 0,Y 124.53,Z 552.629,A -85,B 0,C 180,E1 -25635.171,E2 -25635.171} C_VEL
LIN {X 0,Y 123.792,Z 563.229,A -85,B 0,C 180,E1 -25639.368,E2 -25639.368} C_VEL
LIN {X 0,Y 123.477,Z 571.774,A -85,B 0,C 180,E1 -25643.464,E2 -25643.464} C_VEL
LIN {X 0,Y 123.626,Z 578.927,A -85,B 0,C 180,E1 -25647.557,E2 -25647.557} C_VEL
LIN {X 0,Y 123.762,Z 584.693,A -85,B 0,C 180,E1 -25651.628,E2 -25651.628} C_VEL
LIN {X 0,Y 123.373,Z 588.325,A -85,B 0,C 180,E1 -25654.903,E2 -25654.903} C_VEL
LIN {X 0,Y 122.815,Z 592.737,A -85,B 0,C 180,E1 -25659.886,E2 -25659.886} C_VEL
LIN {X 0,Y 123.511,Z 597.358,A -85,B 0,C 180,E1 -25666.53,E2 -25666.53} C_VEL
LIN {X 0,Y 126.111,Z 600.853,A -85,B 0,C 180,E1 -25672.962,E2 -25672.962} C_VEL
LIN {X 0,Y 130.646,Z 603.401,A -85,B 0,C 180,E1 -25678.957,E2 -25678.957} C_VEL
LIN {X 0,Y 139.148,Z 605.303,A -85,B 0,C 180,E1 -25686.088,E2 -25686.088} C_VEL
LIN {X 0,Y 148.884,Z 605.761,A -85,B 0,C 180,E1 -25691.367,E2 -25691.367} C_VEL
LIN {X 0,Y 158.509,Z 605.198,A -85,B 0,C 180,E1 -25695.188,E2 -25695.188} C_VEL
LIN {X 0,Y 163.707,Z 604.581,A -85,B 0,C 180,E1 -25696.872,E2 -25696.872} C_VEL
LIN {X 0,Y 159.307,Z 604.417,A -85,B 0,C 180,E1 -25698.568,E2 -25698.568} C_VEL
LIN {X 0,Y 149.755,Z 603.407,A -85,B 0,C 180,E1 -25702.405,E2 -25702.405} C_VEL
LIN {X 0,Y 141.269,Z 601.366,A -85,B 0,C 180,E1 -25706.823,E2 -25706.823} C_VEL
LIN {X 0,Y 134.136,Z 598.291,A -85,B 0,C 180,E1 -25711.866,E2 -25711.866} C_VEL
LIN {X 0,Y 128.547,Z 594.175,A -85,B 0,C 180,E1 -25717.499,E2 -25717.499} C_VEL
LIN {X 0,Y 123.868,Z 587.815,A -85,B 0,C 180,E1 -25724.699,E2 -25724.699} C_VEL
LIN {X 0,Y 121.874,Z 580.389,A -85,B 0,C 180,E1 -25731.712,E2 -25731.712} C_VEL
LIN {X 0,Y 121.151,Z 572.922,A -85,B 0,C 180,E1 -25737.507,E2 -25737.507} C_VEL
LIN {X 0,Y 121.151,Z 568.402,A -85,B 0,C 180,E1 -25740.497,E2 -25740.497} C_VEL
LIN {X 0,Y 120.523,Z 564.621,A -85,B 0,C 180,E1 -25742.624,E2 -25742.624} C_VEL
LIN {X 0,Y 117.987,Z 557.698,A -85,B 0,C 180,E1 -25745.812,E2 -25745.812} C_VEL
LIN {X 0,Y 115.674,Z 550.297,A -85,B 0,C 180,E1 -25748.91,E2 -25748.91} C_VEL
LIN {X 0,Y 115.466,Z 545.717,A -85,B 0,C 180,E1 -25750.819,E2 -25750.819} C_VEL
LIN {X 0,Y 116.824,Z 532.779,A -85,B 0,C 180,E1 -25755.729,E2 -25755.729} C_VEL
LIN {X 0,Y 117.886,Z 523.033,A -85,B 0,C 180,E1 -25758.69,E2 -25758.69} C_VEL
LIN {X 0,Y 115.274,Z 509.185,A -85,B 0,C 180,E1 -25761.88,E2 -25761.88} C_VEL
LIN {X 0,Y 114.079,Z 502.272,A -85,B 0,C 180,E1 -25763.273,E2 -25763.273} C_VEL
LIN {X 0,Y 114.133,Z 502.266,A -85,B 0,C 180,E1 -25770.447,E2 -25770.447} C_VEL
LIN {X 0,Y 114.588,Z 502.211,A -85,B 0,C 180,E1 -25777.123,E2 -25777.123} C_VEL
LIN {X 0,Y 114.73,Z 502.188,A -85,B 0,C 180,E1 -25782.685,E2 -25782.685} C_VEL
LIN {X 0,Y 114.804,Z 502.184,A -85,B 0,C 180,E1 -25787.669,E2 -25787.669} C_VEL
LIN {X 0,Y 114.816,Z 502.182,A -85,B 0,C 180,E1 -25792.727,E2 -25792.727} C_VEL
LIN {X 0,Y 114.873,Z 502.168,A -85,B 0,C 180,E1 -25798.932,E2 -25798.932} C_VEL
LIN {X 0,Y 114.951,Z 502.161,A -85,B 0,C 180,E1 -25806.507,E2 -25806.507} C_VEL
LIN {X 0,Y 115.015,Z 502.159,A -85,B 0,C 180,E1 -25812.209,E2 -25812.209} C_VEL
LIN {X 0,Y 115.256,Z 502.121,A -85,B 0,C 180,E1 -25817.333,E2 -25817.333} C_VEL
LIN {X 0,Y 115.37,Z 502.112,A -85,B 0,C 180,E1 -25823.001,E2 -25823.001} C_VEL
LIN {X 0,Y 115.996,Z 502.037,A -85,B 0,C 180,E1 -25829.999,E2 -25829.999} C_VEL
LIN {X 0,Y 115.367,Z 502.112,A -85,B 0,C 180,E1 -25836.997,E2 -25836.997} C_VEL
LIN {X 0,Y 115.255,Z 502.121,A -85,B 0,C 180,E1 -25842.665,E2 -25842.665} C_VEL
LIN {X 0,Y 115.014,Z 502.159,A -85,B 0,C 180,E1 -25847.789,E2 -25847.789} C_VEL
LIN {X 0,Y 114.949,Z 502.162,A -85,B 0,C 180,E1 -25853.491,E2 -25853.491} C_VEL
LIN {X 0,Y 114.871,Z 502.168,A -85,B 0,C 180,E1 -25861.067,E2 -25861.067} C_VEL
LIN {X 0,Y 114.804,Z 502.181,A -85,B 0,C 180,E1 -25867.746,E2 -25867.746} C_VEL
LIN {X 0,Y 114.796,Z 502.184,A -85,B 0,C 180,E1 -25872.72,E2 -25872.72} C_VEL
LIN {X 0,Y 114.796,Z 502.179,A -85,B 0,C 180,E1 -25877.665,E2 -25877.665} C_VEL
LIN {X 0,Y 114.789,Z 502.186,A -85,B 0,C 180,E1 -25882.742,E2 -25882.742} C_VEL
LIN {X 0,Y 114.862,Z 502.174,A -85,B 0,C 180,E1 -25888.937,E2 -25888.937} C_VEL
LIN {X 0,Y 114.947,Z 502.16,A -85,B 0,C 180,E1 -25896.506,E2 -25896.506} C_VEL
LIN {X 0,Y 115.015,Z 502.156,A -85,B 0,C 180,E1 -25902.209,E2 -25902.209} C_VEL
LIN {X 0,Y 115.286,Z 502.122,A -85,B 0,C 180,E1 -25907.257,E2 -25907.257} C_VEL
LIN {X 0,Y 115.393,Z 502.112,A -85,B 0,C 180,E1 -25909.471,E2 -25909.471} C_VEL
LIN {X 0,Y 115.538,Z 502.092,A -85,B 0,C 180,E1 -25916.512,E2 -25916.512} C_VEL
LIN {X 0,Y 115.996,Z 502.033,A -85,B 0,C 180,E1 -25919.999,E2 -25919.999} C_VEL
LIN {X 0,Y 115.398,Z 502.111,A -85,B 0,C 180,E1 -25926.995,E2 -25926.995} C_VEL
LIN {X 0,Y 115.393,Z 502.104,A -85,B 0,C 180,E1 -25930.527,E2 -25930.527} C_VEL
LIN {X 0,Y 115.149,Z 502.141,A -85,B 0,C 180,E1 -25934.13,E2 -25934.13} C_VEL
LIN {X 0,Y 114.982,Z 502.159,A -85,B 0,C 180,E1 -25941.514,E2 -25941.514} C_VEL
LIN {X 0,Y 114.87,Z 502.176,A -85,B 0,C 180,E1 -25945.357,E2 -25945.357} C_VEL
LIN {X 0,Y 114.869,Z 502.174,A -85,B 0,C 180,E1 -25951.069,E2 -25951.069} C_VEL
LIN {X 0,Y 114.937,Z 502.161,A -85,B 0,C 180,E1 -25957.695,E2 -25957.695} C_VEL
LIN {X 0,Y 115.17,Z 502.139,A -85,B 0,C 180,E1 -25962.924,E2 -25962.924} C_VEL
LIN {X 0,Y 115.598,Z 502.085,A -85,B 0,C 180,E1 -25968.029,E2 -25968.029} C_VEL
LIN {X 0,Y 115.898,Z 502.05,A -85,B 0,C 180,E1 -25972.672,E2 -25972.672} C_VEL
LIN {X 0,Y 115.516,Z 502.237,A -85,B 0,C 180,E1 -25974.692,E2 -25974.692} C_VEL
LIN {X 0,Y 114.262,Z 505.204,A -85,B 0,C 180,E1 -25980.525,E2 -25980.525} C_VEL
LIN {X 0,Y 113.81,Z 507.45,A -85,B 0,C 180,E1 -25985.052,E2 -25985.052} C_VEL
LIN {X 0,Y 114.062,Z 522.403,A -85,B 0,C 180,E1 -25987.93,E2 -25987.93} C_VEL
LIN {X 0,Y 115.273,Z 536.462,A -85,B 0,C 180,E1 -25991.333,E2 -25991.333} C_VEL
LIN {X 0,Y 116.989,Z 548.529,A -85,B 0,C 180,E1 -25994.879,E2 -25994.879} C_VEL
LIN {X 0,Y 117.616,Z 552.444,A -85,B 0,C 180,E1 -25996.172,E2 -25996.172} C_VEL
LIN {X 0,Y 116.987,Z 562.67,A -85,B 0,C 180,E1 -26000.492,E2 -26000.492} C_VEL
LIN {X 0,Y 116.807,Z 571.013,A -85,B 0,C 180,E1 -26004.823,E2 -26004.823} C_VEL
LIN {X 0,Y 117.075,Z 578.038,A -85,B 0,C 180,E1 -26009.141,E2 -26009.141} C_VEL
LIN {X 0,Y 117.188,Z 582.689,A -85,B 0,C 180,E1 -26012.579,E2 -26012.579} C_VEL
LIN {X 0,Y 116.618,Z 587.138,A -85,B 0,C 180,E1 -26016.923,E2 -26016.923} C_VEL
LIN {X 0,Y 116.485,Z 592.717,A -85,B 0,C 180,E1 -26023.966,E2 -26023.966} C_VEL
LIN {X 0,Y 118.227,Z 597.021,A -85,B 0,C 180,E1 -26030.897,E2 -26030.897} C_VEL
LIN {X 0,Y 122.071,Z 600.362,A -85,B 0,C 180,E1 -26037.426,E2 -26037.426} C_VEL
LIN {X 0,Y 127.687,Z 602.755,A -85,B 0,C 180,E1 -26043.396,E2 -26043.396} C_VEL
LIN {X 0,Y 134.914,Z 604.24,A -85,B 0,C 180,E1 -26048.691,E2 -26048.691} C_VEL
LIN {X 0,Y 143.672,Z 604.923,A -85,B 0,C 180,E1 -26053.224,E2 -26053.224} C_VEL
LIN {X 0,Y 152.081,Z 604.864,A -85,B 0,C 180,E1 -26056.527,E2 -26056.527} C_VEL
LIN {X 0,Y 152.351,Z 604.672,A -85,B 0,C 180,E1 -26057.426,E2 -26057.426} C_VEL
LIN {X 0,Y 144.208,Z 603.382,A -85,B 0,C 180,E1 -26060.688,E2 -26060.688} C_VEL
LIN {X 0,Y 135.406,Z 600.919,A -85,B 0,C 180,E1 -26065.185,E2 -26065.185} C_VEL
LIN {X 0,Y 126.381,Z 596.444,A -85,B 0,C 180,E1 -26071.792,E2 -26071.792} C_VEL
LIN {X 0,Y 120.891,Z 591.667,A -85,B 0,C 180,E1 -26077.799,E2 -26077.799} C_VEL
LIN {X 0,Y 116.792,Z 585.043,A -85,B 0,C 180,E1 -26084.913,E2 -26084.913} C_VEL
LIN {X 0,Y 115.119,Z 578.324,A -85,B 0,C 180,E1 -26091.222,E2 -26091.222} C_VEL
LIN {X 0,Y 114.424,Z 570.392,A -85,B 0,C 180,E1 -26097.361,E2 -26097.361} C_VEL
LIN {X 0,Y 114.393,Z 562.195,A -85,B 0,C 180,E1 -26102.642,E2 -26102.642} C_VEL
LIN {X 0,Y 114.779,Z 553.973,A -85,B 0,C 180,E1 -26107.035,E2 -26107.035} C_VEL
LIN {X 0,Y 115.466,Z 545.717,A -85,B 0,C 180,E1 -26110.819,E2 -26110.819} C_VEL
LIN {X 0,Y 115.468,Z 541.105,A -85,B 0,C 180,E1 -26112.642,E2 -26112.642} C_VEL
LIN {X 0,Y 114.695,Z 536.229,A -85,B 0,C 180,E1 -26114.311,E2 -26114.311} C_VEL
LIN {X 0,Y 111.93,Z 526.112,A -85,B 0,C 180,E1 -26117.303,E2 -26117.303} C_VEL
LIN {X 0,Y 110.068,Z 519.082,A -85,B 0,C 180,E1 -26119.106,E2 -26119.106} C_VEL
LIN {X 0,Y 107.318,Z 504.352,A -85,B 0,C 180,E1 -26122.439,E2 -26122.439} C_VEL
LIN {X 0,Y 107.105,Z 503.141,A -85,B 0,C 180,E1 -26122.805,E2 -26122.805} C_VEL
LIN {X 0,Y 107.121,Z 503.137,A -85,B 0,C 180,E1 -26131.66,E2 -26131.66} C_VEL
LIN {X 0,Y 107.437,Z 503.101,A -85,B 0,C 180,E1 -26136.069,E2 -26136.069} C_VEL
LIN {X 0,Y 107.565,Z 503.079,A -85,B 0,C 180,E1 -26140.798,E2 -26140.798} C_VEL
LIN {X 0,Y 107.669,Z 503.073,A -85,B 0,C 180,E1 -26145.893,E2 -26145.893} C_VEL
LIN {X 0,Y 107.71,Z 503.062,A -85,B 0,C 180,E1 -26151.537,E2 -26151.537} C_VEL
LIN {X 0,Y 107.811,Z 503.048,A -85,B 0,C 180,E1 -26158.566,E2 -26158.566} C_VEL
LIN {X 0,Y 107.914,Z 503.037,A -85,B 0,C 180,E1 -26166.998,E2 -26166.998} C_VEL
LIN {X 0,Y 108.034,Z 503.024,A -85,B 0,C 180,E1 -26174.916,E2 -26174.916} C_VEL
LIN {X 0,Y 108.257,Z 502.998,A -85,B 0,C 180,E1 -26178.769,E2 -26178.769} C_VEL
LIN {X 0,Y 108.451,Z 502.969,A -85,B 0,C 180,E1 -26186.284,E2 -26186.284} C_VEL
LIN {X 0,Y 108.946,Z 502.915,A -85,B 0,C 180,E1 -26189.999,E2 -26189.999} C_VEL
LIN {X 0,Y 108.306,Z 502.993,A -85,B 0,C 180,E1 -26197.456,E2 -26197.456} C_VEL
LIN {X 0,Y 108.176,Z 503.002,A -85,B 0,C 180,E1 -26202.954,E2 -26202.954} C_VEL
LIN {X 0,Y 107.907,Z 503.042,A -85,B 0,C 180,E1 -26209.004,E2 -26209.004} C_VEL
LIN {X 0,Y 107.86,Z 503.047,A -85,B 0,C 180,E1 -26214.184,E2 -26214.184} C_VEL
LIN {X 0,Y 107.797,Z 503.052,A -85,B 0,C 180,E1 -26222.051,E2 -26222.051} C_VEL
LIN {X 0,Y 107.709,Z 503.062,A -85,B 0,C 180,E1 -26228.462,E2 -26228.462} C_VEL
LIN {X 0,Y 107.68,Z 503.069,A -85,B 0,C 180,E1 -26235.884,E2 -26235.884} C_VEL
LIN {X 0,Y 107.689,Z 503.07,A -85,B 0,C 180,E1 -26241.548,E2 -26241.548} C_VEL
LIN {X 0,Y 107.797,Z 503.053,A -85,B 0,C 180,E1 -26248.561,E2 -26248.561} C_VEL
LIN {X 0,Y 107.911,Z 503.037,A -85,B 0,C 180,E1 -26256.997,E2 -26256.997} C_VEL
LIN {X 0,Y 108.038,Z 503.019,A -85,B 0,C 180,E1 -26264.917,E2 -26264.917} C_VEL
LIN {X 0,Y 108.306,Z 502.993,A -85,B 0,C 180,E1 -26268.774,E2 -26268.774} C_VEL
LIN {X 0,Y 108.464,Z 502.973,A -85,B 0,C 180,E1 -26276.284,E2 -26276.284} C_VEL
LIN {X 0,Y 108.947,Z 502.911,A -85,B 0,C 180,E1 -26279.999,E2 -26279.999} C_VEL
LIN {X 0,Y 108.34,Z 502.99,A -85,B 0,C 180,E1 -26287.454,E2 -26287.454} C_VEL
LIN {X 0,Y 108.203,Z 503.003,A -85,B 0,C 180,E1 -26293.025,E2 -26293.025} C_VEL
LIN {X 0,Y 107.91,Z 503.037,A -85,B 0,C 180,E1 -26299.004,E2 -26299.004} C_VEL
LIN {X 0,Y 107.857,Z 503.049,A -85,B 0,C 180,E1 -26304.184,E2 -26304.184} C_VEL
LIN {X 0,Y 107.801,Z 503.056,A -85,B 0,C 180,E1 -26312.058,E2 -26312.058} C_VEL
LIN {X 0,Y 107.874,Z 503.042,A -85,B 0,C 180,E1 -26318.575,E2 -26318.575} C_VEL
LIN {X 0,Y 108.286,Z 502.994,A -85,B 0,C 180,E1 -26325.554,E2 -26325.554} C_VEL
LIN {X 0,Y 108.74,Z 502.941,A -85,B 0,C 180,E1 -26330.856,E2 -26330.856} C_VEL
LIN {X 0,Y 108.479,Z 502.974,A -85,B 0,C 180,E1 -26334.333,E2 -26334.333} C_VEL
LIN {X 0,Y 107.865,Z 503.134,A -85,B 0,C 180,E1 -26336.954,E2 -26336.954} C_VEL
LIN {X 0,Y 106.759,Z 507.004,A -85,B 0,C 180,E1 -26345.317,E2 -26345.317} C_VEL
LIN {X 0,Y 107.023,Z 521.457,A -85,B 0,C 180,E1 -26348.323,E2 -26348.323} C_VEL
LIN {X 0,Y 108.262,Z 535.479,A -85,B 0,C 180,E1 -26351.935,E2 -26351.935} C_VEL
LIN {X 0,Y 110.09,Z 547.558,A -85,B 0,C 180,E1 -26355.679,E2 -26355.679} C_VEL
LIN {X 0,Y 110.753,Z 551.777,A -85,B 0,C 180,E1 -26357.169,E2 -26357.169} C_VEL
LIN {X 0,Y 110.277,Z 561.808,A -85,B 0,C 180,E1 -26361.757,E2 -26361.757} C_VEL
LIN {X 0,Y 110.277,Z 570.17,A -85,B 0,C 180,E1 -26366.347,E2 -26366.347} C_VEL
LIN {X 0,Y 110.591,Z 577.129,A -85,B 0,C 180,E1 -26370.911,E2 -26370.911} C_VEL
LIN {X 0,Y 110.711,Z 580.544,A -85,B 0,C 180,E1 -26373.64,E2 -26373.64} C_VEL
LIN {X 0,Y 110.035,Z 585.808,A -85,B 0,C 180,E1 -26379.189,E2 -26379.189} C_VEL
LIN {X 0,Y 110.122,Z 590.066,A -85,B 0,C 180,E1 -26384.791,E2 -26384.791} C_VEL
LIN {X 0,Y 112.004,Z 594.679,A -85,B 0,C 180,E1 -26392.117,E2 -26392.117} C_VEL
LIN {X 0,Y 116.074,Z 598.281,A -85,B 0,C 180,E1 -26398.973,E2 -26398.973} C_VEL
LIN {X 0,Y 122.001,Z 600.979,A -85,B 0,C 180,E1 -26405.175,E2 -26405.175} C_VEL
LIN {X 0,Y 129.55,Z 602.841,A -85,B 0,C 180,E1 -26410.617,E2 -26410.617} C_VEL
LIN {X 0,Y 140.828,Z 604.022,A -85,B 0,C 180,E1 -26416.115,E2 -26416.115} C_VEL
LIN {X 0,Y 141.943,Z 604.065,A -85,B 0,C 180,E1 -26416.554,E2 -26416.554} C_VEL
LIN {X 0,Y 140.984,Z 603.661,A -85,B 0,C 180,E1 -26417.899,E2 -26417.899} C_VEL
LIN {X 0,Y 129.669,Z 600.282,A -85,B 0,C 180,E1 -26423.403,E2 -26423.403} C_VEL
LIN {X 0,Y 120.27,Z 595.3,A -85,B 0,C 180,E1 -26430.219,E2 -26430.219} C_VEL
LIN {X 0,Y 114.515,Z 590.106,A -85,B 0,C 180,E1 -26436.49,E2 -26436.49} C_VEL
LIN {X 0,Y 110.697,Z 584.295,A -85,B 0,C 180,E1 -26442.786,E2 -26442.786} C_VEL
LIN {X 0,Y 108.617,Z 577.081,A -85,B 0,C 180,E1 -26449.751,E2 -26449.751} C_VEL
LIN {X 0,Y 107.816,Z 570.237,A -85,B 0,C 180,E1 -26455.327,E2 -26455.327} C_VEL
LIN {X 0,Y 107.661,Z 562.064,A -85,B 0,C 180,E1 -26460.936,E2 -26460.936} C_VEL
LIN {X 0,Y 107.903,Z 554.013,A -85,B 0,C 180,E1 -26465.608,E2 -26465.608} C_VEL
LIN {X 0,Y 108.656,Z 543.344,A -85,B 0,C 180,E1 -26470.718,E2 -26470.718} C_VEL
LIN {X 0,Y 109.962,Z 530.684,A -85,B 0,C 180,E1 -26475.601,E2 -26475.601} C_VEL
LIN {X 0,Y 110.821,Z 523.007,A -85,B 0,C 180,E1 -26478.075,E2 -26478.075} C_VEL
LIN {X 0,Y 110.068,Z 519.082,A -85,B 0,C 180,E1 -26479.106,E2 -26479.106} C_VEL
LIN {X 0,Y 108.908,Z 516.909,A -85,B 0,C 180,E1 -26479.576,E2 -26479.576} C_VEL
LIN {X 0,Y 102.186,Z 511.045,A -85,B 0,C 180,E1 -26480.515,E2 -26480.515} C_VEL
LIN {X 0,Y 101.06,Z 508.808,A -85,B 0,C 180,E1 -26480.957,E2 -26480.957} C_VEL
LIN {X 0,Y 100.14,Z 504.01,A -85,B 0,C 180,E1 -26482.134,E2 -26482.134} C_VEL
LIN {X 0,Y 100.099,Z 504.008,A -85,B 0,C 180,E1 -26492.591,E2 -26492.591} C_VEL
LIN {X 0,Y 100.487,Z 503.965,A -85,B 0,C 180,E1 -26499.704,E2 -26499.704} C_VEL
LIN {X 0,Y 100.635,Z 503.949,A -85,B 0,C 180,E1 -26505.702,E2 -26505.702} C_VEL
LIN {X 0,Y 100.647,Z 503.941,A -85,B 0,C 180,E1 -26511.063,E2 -26511.063} C_VEL
LIN {X 0,Y 100.704,Z 503.938,A -85,B 0,C 180,E1 -26516.876,E2 -26516.876} C_VEL
LIN {X 0,Y 100.789,Z 503.929,A -85,B 0,C 180,E1 -26525.267,E2 -26525.267} C_VEL
LIN {X 0,Y 100.819,Z 503.922,A -85,B 0,C 180,E1 -26529.601,E2 -26529.601} C_VEL
LIN {X 0,Y 101.106,Z 503.882,A -85,B 0,C 180,E1 -26536.701,E2 -26536.701} C_VEL
LIN {X 0,Y 101.247,Z 503.873,A -85,B 0,C 180,E1 -26542.019,E2 -26542.019} C_VEL
LIN {X 0,Y 101.869,Z 503.797,A -85,B 0,C 180,E1 -26549.999,E2 -26549.999} C_VEL
LIN {X 0,Y 101.244,Z 503.874,A -85,B 0,C 180,E1 -26557.979,E2 -26557.979} C_VEL
LIN {X 0,Y 101.105,Z 503.882,A -85,B 0,C 180,E1 -26563.297,E2 -26563.297} C_VEL
LIN {X 0,Y 100.818,Z 503.922,A -85,B 0,C 180,E1 -26570.398,E2 -26570.398} C_VEL
LIN {X 0,Y 100.776,Z 503.93,A -85,B 0,C 180,E1 -26574.957,E2 -26574.957} C_VEL
LIN {X 0,Y 100.702,Z 503.939,A -85,B 0,C 180,E1 -26583.123,E2 -26583.123} C_VEL
LIN {X 0,Y 100.656,Z 503.939,A -85,B 0,C 180,E1 -26589.819,E2 -26589.819} C_VEL
LIN {X 0,Y 100.651,Z 503.945,A -85,B 0,C 180,E1 -26595.711,E2 -26595.711} C_VEL
LIN {X 0,Y 100.628,Z 503.948,A -85,B 0,C 180,E1 -26601.054,E2 -26601.054} C_VEL
LIN {X 0,Y 100.691,Z 503.934,A -85,B 0,C 180,E1 -26606.883,E2 -26606.883} C_VEL
LIN {X 0,Y 100.786,Z 503.923,A -85,B 0,C 180,E1 -26615.266,E2 -26615.266} C_VEL
LIN {X 0,Y 100.817,Z 503.927,A -85,B 0,C 180,E1 -26619.6,E2 -26619.6} C_VEL
LIN {X 0,Y 101.199,Z 503.879,A -85,B 0,C 180,E1 -26627.974,E2 -26627.974} C_VEL
LIN {X 0,Y 101.28,Z 503.864,A -85,B 0,C 180,E1 -26632.022,E2 -26632.022} C_VEL
LIN {X 0,Y 101.871,Z 503.792,A -85,B 0,C 180,E1 -26639.999,E2 -26639.999} C_VEL
LIN {X 0,Y 101.279,Z 503.868,A -85,B 0,C 180,E1 -26647.977,E2 -26647.977} C_VEL
LIN {X 0,Y 101.129,Z 503.885,A -85,B 0,C 180,E1 -26653.363,E2 -26653.363} C_VEL
LIN {X 0,Y 100.819,Z 503.919,A -85,B 0,C 180,E1 -26660.398,E2 -26660.398} C_VEL
LIN {X 0,Y 100.773,Z 503.933,A -85,B 0,C 180,E1 -26664.958,E2 -26664.958} C_VEL
LIN {X 0,Y 100.716,Z 503.94,A -85,B 0,C 180,E1 -26673.138,E2 -26673.138} C_VEL
LIN {X 0,Y 100.881,Z 503.918,A -85,B 0,C 180,E1 -26679.976,E2 -26679.976} C_VEL
LIN {X 0,Y 101.253,Z 503.868,A -85,B 0,C 180,E1 -26686.045,E2 -26686.045} C_VEL
LIN {X 0,Y 101.605,Z 503.83,A -85,B 0,C 180,E1 -26691.5,E2 -26691.5} C_VEL
LIN {X 0,Y 100.787,Z 503.927,A -85,B 0,C 180,E1 -26696.8,E2 -26696.8} C_VEL
LIN {X 0,Y 100.141,Z 504.175,A -85,B 0,C 180,E1 -26700.084,E2 -26700.084} C_VEL
LIN {X 0,Y 99.738,Z 506.629,A -85,B 0,C 180,E1 -26705.836,E2 -26705.836} C_VEL
LIN {X 0,Y 100.051,Z 520.832,A -85,B 0,C 180,E1 -26708.995,E2 -26708.995} C_VEL
LIN {X 0,Y 101.383,Z 534.927,A -85,B 0,C 180,E1 -26712.866,E2 -26712.866} C_VEL
LIN {X 0,Y 103.275,Z 546.686,A -85,B 0,C 180,E1 -26716.723,E2 -26716.723} C_VEL
LIN {X 0,Y 103.963,Z 550.903,A -85,B 0,C 180,E1 -26718.3,E2 -26718.3} C_VEL
LIN {X 0,Y 103.616,Z 560.932,A -85,B 0,C 180,E1 -26723.184,E2 -26723.184} C_VEL
LIN {X 0,Y 103.805,Z 569.225,A -85,B 0,C 180,E1 -26728.061,E2 -26728.061} C_VEL
LIN {X 0,Y 104.294,Z 576.01,A -85,B 0,C 180,E1 -26732.898,E2 -26732.898} C_VEL
LIN {X 0,Y 104.147,Z 579.22,A -85,B 0,C 180,E1 -26735.81,E2 -26735.81} C_VEL
LIN {X 0,Y 103.61,Z 584.33,A -85,B 0,C 180,E1 -26741.742,E2 -26741.742} C_VEL
LIN {X 0,Y 104.607,Z 589.95,A -85,B 0,C 180,E1 -26749.851,E2 -26749.851} C_VEL
LIN {X 0,Y 107.785,Z 594.18,A -85,B 0,C 180,E1 -26757.158,E2 -26757.158} C_VEL
LIN {X 0,Y 113.138,Z 597.639,A -85,B 0,C 180,E1 -26763.992,E2 -26763.992} C_VEL
LIN {X 0,Y 120.246,Z 600.232,A -85,B 0,C 180,E1 -26770.011,E2 -26770.011} C_VEL
LIN {X 0,Y 130.978,Z 602.299,A -85,B 0,C 180,E1 -26776.067,E2 -26776.067} C_VEL
LIN {X 0,Y 132.066,Z 602.246,A -85,B 0,C 180,E1 -26777.474,E2 -26777.474} C_VEL
LIN {X 0,Y 124.094,Z 599.401,A -85,B 0,C 180,E1 -26781.467,E2 -26781.467} C_VEL
LIN {X 0,Y 116.007,Z 595.144,A -85,B 0,C 180,E1 -26786.96,E2 -26786.96} C_VEL
LIN {X 0,Y 109.589,Z 589.902,A -85,B 0,C 180,E1 -26793.327,E2 -26793.327} C_VEL
LIN {X 0,Y 104.245,Z 582.206,A -85,B 0,C 180,E1 -26801.665,E2 -26801.665} C_VEL
LIN {X 0,Y 102.042,Z 574.579,A -85,B 0,C 180,E1 -26809.083,E2 -26809.083} C_VEL
LIN {X 0,Y 101.116,Z 566.125,A -85,B 0,C 180,E1 -26816.015,E2 -26816.015} C_VEL
LIN {X 0,Y 101.016,Z 557.168,A -85,B 0,C 180,E1 -26821.994,E2 -26821.994} C_VEL
LIN {X 0,Y 101.513,Z 546.306,A -85,B 0,C 180,E1 -26827.96,E2 -26827.96} C_VEL
LIN {X 0,Y 102.389,Z 535.345,A -85,B 0,C 180,E1 -26832.891,E2 -26832.891} C_VEL
LIN {X 0,Y 103.665,Z 523.383,A -85,B 0,C 180,E1 -26837.19,E2 -26837.19} C_VEL
LIN {X 0,Y 103.436,Z 520.736,A -85,B 0,C 180,E1 -26837.963,E2 -26837.963} C_VEL
LIN {X 0,Y 101.06,Z 508.808,A -85,B 0,C 180,E1 -26840.957,E2 -26840.957} C_VEL
LIN {X 0,Y 100.208,Z 506.546,A -85,B 0,C 180,E1 -26841.954,E2 -26841.954} C_VEL
LIN {X 0,Y 98.719,Z 504.993,A -85,B 0,C 180,E1 -26843.877,E2 -26843.877} C_VEL
LIN {X 0,Y 97.308,Z 504.51,A -85,B 0,C 180,E1 -26845.961,E2 -26845.961} C_VEL
LIN {X 0,Y 93.391,Z 504.851,A -85,B 0,C 180,E1 -26856.171,E2 -26856.171} C_VEL
LIN {X 0,Y 93.261,Z 504.857,A -85,B 0,C 180,E1 -26858.94,E2 -26858.94} C_VEL
LIN {X 0,Y 93.445,Z 504.838,A -85,B 0,C 180,E1 -26862.603,E2 -26862.603} C_VEL
LIN {X 0,Y 93.542,Z 504.829,A -85,B 0,C 180,E1 -26868.707,E2 -26868.707} C_VEL
LIN {X 0,Y 93.602,Z 504.826,A -85,B 0,C 180,E1 -26875.685,E2 -26875.685} C_VEL
LIN {X 0,Y 93.673,Z 504.817,A -85,B 0,C 180,E1 -26884.204,E2 -26884.204} C_VEL
LIN {X 0,Y 93.696,Z 504.806,A -85,B 0,C 180,E1 -26887.972,E2 -26887.972} C_VEL
LIN {X 0,Y 94.026,Z 504.764,A -85,B 0,C 180,E1 -26896.341,E2 -26896.341} C_VEL
LIN {X 0,Y 94.18,Z 504.754,A -85,B 0,C 180,E1 -26901.416,E2 -26901.416} C_VEL
LIN {X 0,Y 94.794,Z 504.678,A -85,B 0,C 180,E1 -26909.999,E2 -26909.999} C_VEL
LIN {X 0,Y 94.178,Z 504.754,A -85,B 0,C 180,E1 -26918.583,E2 -26918.583} C_VEL
LIN {X 0,Y 94.025,Z 504.764,A -85,B 0,C 180,E1 -26923.657,E2 -26923.657} C_VEL
LIN {X 0,Y 93.694,Z 504.806,A -85,B 0,C 180,E1 -26932.026,E2 -26932.026} C_VEL
LIN {X 0,Y 93.625,Z 504.822,A -85,B 0,C 180,E1 -26936.768,E2 -26936.768} C_VEL
LIN {X 0,Y 93.6,Z 504.826,A -85,B 0,C 180,E1 -26944.314,E2 -26944.314} C_VEL
LIN {X 0,Y 93.54,Z 504.832,A -85,B 0,C 180,E1 -26952.546,E2 -26952.546} C_VEL
LIN {X 0,Y 93.537,Z 504.825,A -85,B 0,C 180,E1 -26958.707,E2 -26958.707} C_VEL
LIN {X 0,Y 93.588,Z 504.821,A -85,B 0,C 180,E1 -26965.693,E2 -26965.693} C_VEL
LIN {X 0,Y 93.669,Z 504.813,A -85,B 0,C 180,E1 -26974.204,E2 -26974.204} C_VEL
LIN {X 0,Y 93.694,Z 504.811,A -85,B 0,C 180,E1 -26977.971,E2 -26977.971} C_VEL
LIN {X 0,Y 94.098,Z 504.761,A -85,B 0,C 180,E1 -26987.051,E2 -26987.051} C_VEL
LIN {X 0,Y 94.212,Z 504.746,A -85,B 0,C 180,E1 -26991.419,E2 -26991.419} C_VEL
LIN {X 0,Y 94.798,Z 504.673,A -85,B 0,C 180,E1 -26999.999,E2 -26999.999} C_VEL
LIN {X 0,Y 94.211,Z 504.748,A -85,B 0,C 180,E1 -27008.579,E2 -27008.579} C_VEL
LIN {X 0,Y 94.046,Z 504.769,A -85,B 0,C 180,E1 -27013.721,E2 -27013.721} C_VEL
LIN {X 0,Y 93.694,Z 504.812,A -85,B 0,C 180,E1 -27022.026,E2 -27022.026} C_VEL
LIN {X 0,Y 93.623,Z 504.819,A -85,B 0,C 180,E1 -27026.769,E2 -27026.769} C_VEL
LIN {X 0,Y 93.643,Z 504.819,A -85,B 0,C 180,E1 -27034.356,E2 -27034.356} C_VEL
LIN {X 0,Y 93.908,Z 504.787,A -85,B 0,C 180,E1 -27042.341,E2 -27042.341} C_VEL
LIN {X 0,Y 94.336,Z 504.733,A -85,B 0,C 180,E1 -27048.157,E2 -27048.157} C_VEL
LIN {X 0,Y 94.207,Z 504.749,A -85,B 0,C 180,E1 -27053.359,E2 -27053.359} C_VEL
LIN {X 0,Y 93.373,Z 504.855,A -85,B 0,C 180,E1 -27058.206,E2 -27058.206} C_VEL
LIN {X 0,Y 92.647,Z 505.156,A -85,B 0,C 180,E1 -27063.768,E2 -27063.768} C_VEL
LIN {X 0,Y 92.738,Z 506.242,A -85,B 0,C 180,E1 -27066.486,E2 -27066.486} C_VEL
LIN {X 0,Y 93.06,Z 519.387,A -85,B 0,C 180,E1 -27069.557,E2 -27069.557} C_VEL
LIN {X 0,Y 94.254,Z 531.997,A -85,B 0,C 180,E1 -27073.165,E2 -27073.165} C_VEL
LIN {X 0,Y 96.52,Z 545.831,A -85,B 0,C 180,E1 -27077.917,E2 -27077.917} C_VEL
LIN {X 0,Y 97.243,Z 550.022,A -85,B 0,C 180,E1 -27079.591,E2 -27079.591} C_VEL
LIN {X 0,Y 97.098,Z 559.886,A -85,B 0,C 180,E1 -27084.81,E2 -27084.81} C_VEL
LIN {X 0,Y 97.481,Z 568.091,A -85,B 0,C 180,E1 -27090.001,E2 -27090.001} C_VEL
LIN {X 0,Y 97.971,Z 573.584,A -85,B 0,C 180,E1 -27094.115,E2 -27094.115} C_VEL
LIN {X 0,Y 97.908,Z 575.836,A -85,B 0,C 180,E1 -27096.182,E2 -27096.182} C_VEL
LIN {X 0,Y 97.409,Z 581.149,A -85,B 0,C 180,E1 -27102.501,E2 -27102.501} C_VEL
LIN {X 0,Y 98.478,Z 586.943,A -85,B 0,C 180,E1 -27110.907,E2 -27110.907} C_VEL
LIN {X 0,Y 101.944,Z 591.618,A -85,B 0,C 180,E1 -27118.855,E2 -27118.855} C_VEL
LIN {X 0,Y 107.644,Z 595.342,A -85,B 0,C 180,E1 -27125.988,E2 -27125.988} C_VEL
LIN {X 0,Y 115.108,Z 598.219,A -85,B 0,C 180,E1 -27132.193,E2 -27132.193} C_VEL
LIN {X 0,Y 121.777,Z 599.901,A -85,B 0,C 180,E1 -27136.169,E2 -27136.169} C_VEL
LIN {X 0,Y 122.228,Z 599.783,A -85,B 0,C 180,E1 -27137.499,E2 -27137.499} C_VEL
LIN {X 0,Y 112.257,Z 594.898,A -85,B 0,C 180,E1 -27143.505,E2 -27143.505} C_VEL
LIN {X 0,Y 103.514,Z 588,A -85,B 0,C 180,E1 -27151.625,E2 -27151.625} C_VEL
LIN {X 0,Y 98.521,Z 581.151,A -85,B 0,C 180,E1 -27159.105,E2 -27159.105} C_VEL
LIN {X 0,Y 95.771,Z 573.052,A -85,B 0,C 180,E1 -27167.283,E2 -27167.283} C_VEL
LIN {X 0,Y 94.635,Z 564.267,A -85,B 0,C 180,E1 -27174.675,E2 -27174.675} C_VEL
LIN {X 0,Y 94.387,Z 555.22,A -85,B 0,C 180,E1 -27181.068,E2 -27181.068} C_VEL
LIN {X 0,Y 94.819,Z 543.996,A -85,B 0,C 180,E1 -27187.454,E2 -27187.454} C_VEL
LIN {X 0,Y 95.832,Z 531.312,A -85,B 0,C 180,E1 -27193.25,E2 -27193.25} C_VEL
LIN {X 0,Y 96.648,Z 523.064,A -85,B 0,C 180,E1 -27196.368,E2 -27196.368} C_VEL
LIN {X 0,Y 96.272,Z 519.978,A -85,B 0,C 180,E1 -27197.328,E2 -27197.328} C_VEL
LIN {X 0,Y 93.401,Z 505.542,A -85,B 0,C 180,E1 -27201.034,E2 -27201.034} C_VEL
LIN {X 0,Y 93.226,Z 504.874,A -85,B 0,C 180,E1 -27201.342,E2 -27201.342} C_VEL
LIN {X 0,Y 93.112,Z 504.879,A -85,B 0,C 180,E1 -27213.872,E2 -27213.872} C_VEL
LIN {X 0,Y 93.261,Z 504.857,A -85,B 0,C 180,E1 -27218.94,E2 -27218.94} C_VEL
LIN {X 0,Y 93.02,Z 504.89,A -85,B 0,C 180,E1 -27221.349,E2 -27221.349} C_VEL
LIN {X 0,Y 91.752,Z 505.056,A -85,B 0,C 180,E1 -27224.933,E2 -27224.933} C_VEL
LIN {X 0,Y 88.634,Z 505.443,A -85,B 0,C 180,E1 -27231.002,E2 -27231.002} C_VEL
LIN {X 0,Y 86.704,Z 505.684,A -85,B 0,C 180,E1 -27236.184,E2 -27236.184} C_VEL
LIN {X 0,Y 86.414,Z 505.706,A -85,B 0,C 180,E1 -27238.872,E2 -27238.872} C_VEL
LIN {X 0,Y 86.588,Z 505.699,A -85,B 0,C 180,E1 -27243.233,E2 -27243.233} C_VEL
LIN {X 0,Y 86.649,Z 505.691,A -85,B 0,C 180,E1 -27251.067,E2 -27251.067} C_VEL
LIN {X 0,Y 86.934,Z 505.648,A -85,B 0,C 180,E1 -27255.963,E2 -27255.963} C_VEL
LIN {X 0,Y 87.089,Z 505.637,A -85,B 0,C 180,E1 -27260.711,E2 -27260.711} C_VEL
LIN {X 0,Y 87.721,Z 505.559,A -85,B 0,C 180,E1 -27269.999,E2 -27269.999} C_VEL
LIN {X 0,Y 87.087,Z 505.637,A -85,B 0,C 180,E1 -27279.287,E2 -27279.287} C_VEL
LIN {X 0,Y 86.933,Z 505.648,A -85,B 0,C 180,E1 -27284.035,E2 -27284.035} C_VEL
LIN {X 0,Y 86.648,Z 505.691,A -85,B 0,C 180,E1 -27288.931,E2 -27288.931} C_VEL
LIN {X 0,Y 86.587,Z 505.699,A -85,B 0,C 180,E1 -27296.765,E2 -27296.765} C_VEL
LIN {X 0,Y 86.519,Z 505.708,A -85,B 0,C 180,E1 -27305.675,E2 -27305.675} C_VEL
LIN {X 0,Y 86.482,Z 505.712,A -85,B 0,C 180,E1 -27312.995,E2 -27312.995} C_VEL
LIN {X 0,Y 86.458,Z 505.708,A -85,B 0,C 180,E1 -27319.434,E2 -27319.434} C_VEL
LIN {X 0,Y 86.531,Z 505.701,A -85,B 0,C 180,E1 -27325.35,E2 -27325.35} C_VEL
LIN {X 0,Y 86.585,Z 505.698,A -85,B 0,C 180,E1 -27333.233,E2 -27333.233} C_VEL
LIN {X 0,Y 86.663,Z 505.69,A -85,B 0,C 180,E1 -27341.071,E2 -27341.071} C_VEL
LIN {X 0,Y 86.969,Z 505.645,A -85,B 0,C 180,E1 -27345.969,E2 -27345.969} C_VEL
LIN {X 0,Y 87.118,Z 505.632,A -85,B 0,C 180,E1 -27350.714,E2 -27350.714} C_VEL
LIN {X 0,Y 87.725,Z 505.554,A -85,B 0,C 180,E1 -27359.999,E2 -27359.999} C_VEL
LIN {X 0,Y 87.118,Z 505.628,A -85,B 0,C 180,E1 -27369.284,E2 -27369.284} C_VEL
LIN {X 0,Y 86.949,Z 505.654,A -85,B 0,C 180,E1 -27374.086,E2 -27374.086} C_VEL
LIN {X 0,Y 86.587,Z 505.699,A -85,B 0,C 180,E1 -27383.942,E2 -27383.942} C_VEL
LIN {X 0,Y 86.482,Z 505.704,A -85,B 0,C 180,E1 -27389.181,E2 -27389.181} C_VEL
LIN {X 0,Y 86.587,Z 505.694,A -85,B 0,C 180,E1 -27395.742,E2 -27395.742} C_VEL
LIN {X 0,Y 86.894,Z 505.661,A -85,B 0,C 180,E1 -27403.289,E2 -27403.289} C_VEL
LIN {X 0,Y 87.099,Z 505.629,A -85,B 0,C 180,E1 -27406.568,E2 -27406.568} C_VEL
LIN {X 0,Y 87.186,Z 505.626,A -85,B 0,C 180,E1 -27409.845,E2 -27409.845} C_VEL
LIN {X 0,Y 87.107,Z 505.633,A -85,B 0,C 180,E1 -27413.785,E2 -27413.785} C_VEL
LIN {X 0,Y 85.752,Z 505.808,A -85,B 0,C 180,E1 -27427.249,E2 -27427.249} C_VEL
LIN {X 0,Y 86.257,Z 520.246,A -85,B 0,C 180,E1 -27430.98,E2 -27430.98} C_VEL
LIN {X 0,Y 88.024,Z 535.136,A -85,B 0,C 180,E1 -27435.76,E2 -27435.76} C_VEL
LIN {X 0,Y 90.534,Z 547.538,A -85,B 0,C 180,E1 -27440.506,E2 -27440.506} C_VEL
LIN {X 0,Y 90.618,Z 554.984,A -85,B 0,C 180,E1 -27444.438,E2 -27444.438} C_VEL
LIN {X 0,Y 90.972,Z 563.812,A -85,B 0,C 180,E1 -27450.001,E2 -27450.001} C_VEL
LIN {X 0,Y 91.605,Z 569.721,A -85,B 0,C 180,E1 -27454.401,E2 -27454.401} C_VEL
LIN {X 0,Y 91.785,Z 572.168,A -85,B 0,C 180,E1 -27456.596,E2 -27456.596} C_VEL
LIN {X 0,Y 91.319,Z 577.812,A -85,B 0,C 180,E1 -27463.35,E2 -27463.35} C_VEL
LIN {X 0,Y 92.545,Z 583.855,A -85,B 0,C 180,E1 -27472.317,E2 -27472.317} C_VEL
LIN {X 0,Y 96.277,Z 588.818,A -85,B 0,C 180,E1 -27480.731,E2 -27480.731} C_VEL
LIN {X 0,Y 102.332,Z 592.871,A -85,B 0,C 180,E1 -27488.179,E2 -27488.179} C_VEL
LIN {X 0,Y 110.207,Z 596.023,A -85,B 0,C 180,E1 -27494.547,E2 -27494.547} C_VEL
LIN {X 0,Y 113.49,Z 596.958,A -85,B 0,C 180,E1 -27497.064,E2 -27497.064} C_VEL
LIN {X 0,Y 102.794,Z 590.51,A -85,B 0,C 180,E1 -27504.47,E2 -27504.47} C_VEL
LIN {X 0,Y 94.681,Z 582.421,A -85,B 0,C 180,E1 -27513.554,E2 -27513.554} C_VEL
LIN {X 0,Y 90.585,Z 574.575,A -85,B 0,C 180,E1 -27521.921,E2 -27521.921} C_VEL
LIN {X 0,Y 88.678,Z 566.427,A -85,B 0,C 180,E1 -27529.729,E2 -27529.729} C_VEL
LIN {X 0,Y 88.009,Z 557.901,A -85,B 0,C 180,E1 -27536.567,E2 -27536.567} C_VEL
LIN {X 0,Y 87.914,Z 549.453,A -85,B 0,C 180,E1 -27542.292,E2 -27542.292} C_VEL
LIN {X 0,Y 88.267,Z 539.322,A -85,B 0,C 180,E1 -27548.011,E2 -27548.011} C_VEL
LIN {X 0,Y 89.31,Z 526.932,A -85,B 0,C 180,E1 -27553.656,E2 -27553.656} C_VEL
LIN {X 0,Y 89.609,Z 520.893,A -85,B 0,C 180,E1 -27555.934,E2 -27555.934} C_VEL
LIN {X 0,Y 86.536,Z 506.184,A -85,B 0,C 180,E1 -27559.989,E2 -27559.989} C_VEL
LIN {X 0,Y 86.394,Z 505.725,A -85,B 0,C 180,E1 -27560.228,E2 -27560.228} C_VEL
LIN {X 0,Y 85.75,Z 505.803,A -85,B 0,C 180,E1 -27569.458,E2 -27569.458} C_VEL
LIN {X 0,Y 86.1,Z 505.758,A -85,B 0,C 180,E1 -27575.286,E2 -27575.286} C_VEL
LIN {X 0,Y 86.383,Z 505.718,A -85,B 0,C 180,E1 -27582.925,E2 -27582.925} C_VEL
LIN {X 0,Y 86.465,Z 505.708,A -85,B 0,C 180,E1 -27589.438,E2 -27589.438} C_VEL
LIN {X 0,Y 86.546,Z 505.704,A -85,B 0,C 180,E1 -27595.357,E2 -27595.357} C_VEL
LIN {X 0,Y 86.414,Z 505.706,A -85,B 0,C 180,E1 -27598.872,E2 -27598.872} C_VEL
LIN {X 0,Y 85.838,Z 505.793,A -85,B 0,C 180,E1 -27602.771,E2 -27602.771} C_VEL
LIN {X 0,Y 84.43,Z 505.978,A -85,B 0,C 180,E1 -27606.653,E2 -27606.653} C_VEL
LIN {X 0,Y 80.279,Z 506.496,A -85,B 0,C 180,E1 -27617.556,E2 -27617.556} C_VEL
LIN {X 0,Y 79.957,Z 506.519,A -85,B 0,C 180,E1 -27620.455,E2 -27620.455} C_VEL
LIN {X 0,Y 80.647,Z 506.44,A -85,B 0,C 180,E1 -27629.999,E2 -27629.999} C_VEL
LIN {X 0,Y 79.97,Z 506.522,A -85,B 0,C 180,E1 -27640.122,E2 -27640.122} C_VEL
LIN {X 0,Y 79.746,Z 506.548,A -85,B 0,C 180,E1 -27645.329,E2 -27645.329} C_VEL
LIN {X 0,Y 79.515,Z 506.574,A -85,B 0,C 180,E1 -27650.703,E2 -27650.703} C_VEL
LIN {X 0,Y 79.485,Z 506.582,A -85,B 0,C 180,E1 -27657.845,E2 -27657.845} C_VEL
LIN {X 0,Y 79.386,Z 506.589,A -85,B 0,C 180,E1 -27662.084,E2 -27662.084} C_VEL
LIN {X 0,Y 79.374,Z 506.591,A -85,B 0,C 180,E1 -27668.3,E2 -27668.3} C_VEL
LIN {X 0,Y 79.41,Z 506.593,A -85,B 0,C 180,E1 -27675.072,E2 -27675.072} C_VEL
LIN {X 0,Y 79.386,Z 506.596,A -85,B 0,C 180,E1 -27682.82,E2 -27682.82} C_VEL
LIN {X 0,Y 79.378,Z 506.589,A -85,B 0,C 180,E1 -27687.91,E2 -27687.91} C_VEL
LIN {X 0,Y 79.525,Z 506.575,A -85,B 0,C 180,E1 -27693.775,E2 -27693.775} C_VEL
LIN {X 0,Y 79.523,Z 506.579,A -85,B 0,C 180,E1 -27699.296,E2 -27699.296} C_VEL
LIN {X 0,Y 79.841,Z 506.531,A -85,B 0,C 180,E1 -27705.524,E2 -27705.524} C_VEL
LIN {X 0,Y 80,Z 506.519,A -85,B 0,C 180,E1 -27709.879,E2 -27709.879} C_VEL
LIN {X 0,Y 80.653,Z 506.435,A -85,B 0,C 180,E1 -27719.999,E2 -27719.999} C_VEL
LIN {X 0,Y 80,Z 506.512,A -85,B 0,C 180,E1 -27730.118,E2 -27730.118} C_VEL
LIN {X 0,Y 79.762,Z 506.55,A -85,B 0,C 180,E1 -27735.326,E2 -27735.326} C_VEL
LIN {X 0,Y 79.514,Z 506.573,A -85,B 0,C 180,E1 -27740.703,E2 -27740.703} C_VEL
LIN {X 0,Y 79.484,Z 506.575,A -85,B 0,C 180,E1 -27747.848,E2 -27747.848} C_VEL
LIN {X 0,Y 79.534,Z 506.569,A -85,B 0,C 180,E1 -27757.32,E2 -27757.32} C_VEL
LIN {X 0,Y 79.933,Z 506.523,A -85,B 0,C 180,E1 -27765.302,E2 -27765.302} C_VEL
LIN {X 0,Y 80.058,Z 506.513,A -85,B 0,C 180,E1 -27772.191,E2 -27772.191} C_VEL
LIN {X 0,Y 79.218,Z 506.616,A -85,B 0,C 180,E1 -27777.84,E2 -27777.84} C_VEL
LIN {X 0,Y 78.849,Z 506.659,A -85,B 0,C 180,E1 -27788.601,E2 -27788.601} C_VEL
LIN {X 0,Y 79.435,Z 519.716,A -85,B 0,C 180,E1 -27792.298,E2 -27792.298} C_VEL
LIN {X 0,Y 81.143,Z 533.025,A -85,B 0,C 180,E1 -27796.86,E2 -27796.86} C_VEL
LIN {X 0,Y 83.56,Z 544.785,A -85,B 0,C 180,E1 -27801.537,E2 -27801.537} C_VEL
LIN {X 0,Y 84.148,Z 547.554,A -85,B 0,C 180,E1 -27802.804,E2 -27802.804} C_VEL
LIN {X 0,Y 84.373,Z 556.649,A -85,B 0,C 180,E1 -27808.274,E2 -27808.274} C_VEL
LIN {X 0,Y 85.315,Z 565.523,A -85,B 0,C 180,E1 -27814.726,E2 -27814.726} C_VEL
LIN {X 0,Y 85.687,Z 568.263,A -85,B 0,C 180,E1 -27817.068,E2 -27817.068} C_VEL
LIN {X 0,Y 85.439,Z 572.264,A -85,B 0,C 180,E1 -27821.628,E2 -27821.628} C_VEL
LIN {X 0,Y 85.792,Z 577.598,A -85,B 0,C 180,E1 -27829.129,E2 -27829.129} C_VEL
LIN {X 0,Y 88.445,Z 583.331,A -85,B 0,C 180,E1 -27838.476,E2 -27838.476} C_VEL
LIN {X 0,Y 95.461,Z 589.154,A -85,B 0,C 180,E1 -27848.741,E2 -27848.741} C_VEL
LIN {X 0,Y 104.012,Z 593.091,A -85,B 0,C 180,E1 -27856.043,E2 -27856.043} C_VEL
LIN {X 0,Y 103.811,Z 592.782,A -85,B 0,C 180,E1 -27857.391,E2 -27857.391} C_VEL
LIN {X 0,Y 93.804,Z 585.447,A -85,B 0,C 180,E1 -27865.504,E2 -27865.504} C_VEL
LIN {X 0,Y 87.437,Z 577.896,A -85,B 0,C 180,E1 -27873.764,E2 -27873.764} C_VEL
LIN {X 0,Y 83.729,Z 569.345,A -85,B 0,C 180,E1 -27882.917,E2 -27882.917} C_VEL
LIN {X 0,Y 81.998,Z 560.222,A -85,B 0,C 180,E1 -27891.375,E2 -27891.375} C_VEL
LIN {X 0,Y 81.476,Z 552.349,A -85,B 0,C 180,E1 -27897.529,E2 -27897.529} C_VEL
LIN {X 0,Y 81.469,Z 541.891,A -85,B 0,C 180,E1 -27904.33,E2 -27904.33} C_VEL
LIN {X 0,Y 82.092,Z 530.396,A -85,B 0,C 180,E1 -27910.483,E2 -27910.483} C_VEL
LIN {X 0,Y 82.758,Z 522.132,A -85,B 0,C 180,E1 -27914.133,E2 -27914.133} C_VEL
LIN {X 0,Y 82.177,Z 518.464,A -85,B 0,C 180,E1 -27915.372,E2 -27915.372} C_VEL
LIN {X 0,Y 79.619,Z 506.568,A -85,B 0,C 180,E1 -27918.942,E2 -27918.942} C_VEL
LIN {X 0,Y 78.788,Z 506.662,A -85,B 0,C 180,E1 -27932.36,E2 -27932.36} C_VEL
LIN {X 0,Y 79.112,Z 506.629,A -85,B 0,C 180,E1 -27938.454,E2 -27938.454} C_VEL
LIN {X 0,Y 79.331,Z 506.603,A -85,B 0,C 180,E1 -27945.133,E2 -27945.133} C_VEL
LIN {X 0,Y 79.396,Z 506.592,A -85,B 0,C 180,E1 -27952.815,E2 -27952.815} C_VEL
LIN {X 0,Y 79.372,Z 506.588,A -85,B 0,C 180,E1 -27958.855,E2 -27958.855} C_VEL
LIN {X 0,Y 79.529,Z 506.579,A -85,B 0,C 180,E1 -27963.777,E2 -27963.777} C_VEL
LIN {X 0,Y 79.516,Z 506.574,A -85,B 0,C 180,E1 -27969.295,E2 -27969.295} C_VEL
LIN {X 0,Y 79.828,Z 506.534,A -85,B 0,C 180,E1 -27975.572,E2 -27975.572} C_VEL
LIN {X 0,Y 79.957,Z 506.519,A -85,B 0,C 180,E1 -27980.455,E2 -27980.455} C_VEL
LIN {X 0,Y 79.601,Z 506.567,A -85,B 0,C 180,E1 -27983.27,E2 -27983.27} C_VEL
LIN {X 0,Y 78.236,Z 506.735,A -85,B 0,C 180,E1 -27987.461,E2 -27987.461} C_VEL
LIN {X 0,Y 75.056,Z 507.136,A -85,B 0,C 180,E1 -27994.606,E2 -27994.606} C_VEL
LIN {X 0,Y 73.075,Z 507.38,A -85,B 0,C 180,E1 -28000.755,E2 -28000.755} C_VEL
LIN {X 0,Y 72.728,Z 507.417,A -85,B 0,C 180,E1 -28003.957,E2 -28003.957} C_VEL
LIN {X 0,Y 72.396,Z 507.459,A -85,B 0,C 180,E1 -28012.848,E2 -28012.848} C_VEL
LIN {X 0,Y 72.378,Z 507.463,A -85,B 0,C 180,E1 -28019.08,E2 -28019.08} C_VEL
LIN {X 0,Y 72.302,Z 507.479,A -85,B 0,C 180,E1 -28025.676,E2 -28025.676} C_VEL
LIN {X 0,Y 72.262,Z 507.483,A -85,B 0,C 180,E1 -28032.904,E2 -28032.904} C_VEL
LIN {X 0,Y 72.296,Z 507.478,A -85,B 0,C 180,E1 -28041.048,E2 -28041.048} C_VEL
LIN {X 0,Y 72.294,Z 507.478,A -85,B 0,C 180,E1 -28044.316,E2 -28044.316} C_VEL
LIN {X 0,Y 72.375,Z 507.469,A -85,B 0,C 180,E1 -28050.951,E2 -28050.951} C_VEL
LIN {X 0,Y 72.399,Z 507.46,A -85,B 0,C 180,E1 -28057.15,E2 -28057.15} C_VEL
LIN {X 0,Y 72.757,Z 507.412,A -85,B 0,C 180,E1 -28065.001,E2 -28065.001} C_VEL
LIN {X 0,Y 72.885,Z 507.406,A -85,B 0,C 180,E1 -28068.879,E2 -28068.879} C_VEL
LIN {X 0,Y 73.58,Z 507.316,A -85,B 0,C 180,E1 -28079.999,E2 -28079.999} C_VEL
LIN {X 0,Y 72.884,Z 507.397,A -85,B 0,C 180,E1 -28091.118,E2 -28091.118} C_VEL
LIN {X 0,Y 72.582,Z 507.442,A -85,B 0,C 180,E1 -28096.886,E2 -28096.886} C_VEL
LIN {X 0,Y 72.394,Z 507.466,A -85,B 0,C 180,E1 -28102.849,E2 -28102.849} C_VEL
LIN {X 0,Y 72.399,Z 507.458,A -85,B 0,C 180,E1 -28109.115,E2 -28109.115} C_VEL
LIN {X 0,Y 72.494,Z 507.45,A -85,B 0,C 180,E1 -28119.145,E2 -28119.145} C_VEL
LIN {X 0,Y 72.644,Z 507.436,A -85,B 0,C 180,E1 -28122.625,E2 -28122.625} C_VEL
LIN {X 0,Y 72.879,Z 507.408,A -85,B 0,C 180,E1 -28130.485,E2 -28130.485} C_VEL
LIN {X 0,Y 72.551,Z 507.444,A -85,B 0,C 180,E1 -28134.465,E2 -28134.465} C_VEL
LIN {X 0,Y 71.953,Z 507.513,A -85,B 0,C 180,E1 -28150.197,E2 -28150.197} C_VEL
LIN {X 0,Y 73.061,Z 522.459,A -85,B 0,C 180,E1 -28155.073,E2 -28155.073} C_VEL
LIN {X 0,Y 75.169,Z 535.226,A -85,B 0,C 180,E1 -28159.973,E2 -28159.973} C_VEL
LIN {X 0,Y 77.769,Z 546.113,A -85,B 0,C 180,E1 -28164.816,E2 -28164.816} C_VEL
LIN {X 0,Y 78.435,Z 556.547,A -85,B 0,C 180,E1 -28171.695,E2 -28171.695} C_VEL
LIN {X 0,Y 79.57,Z 564.381,A -85,B 0,C 180,E1 -28177.903,E2 -28177.903} C_VEL
LIN {X 0,Y 79.658,Z 566.585,A -85,B 0,C 180,E1 -28180.164,E2 -28180.164} C_VEL
LIN {X 0,Y 80.043,Z 573.992,A -85,B 0,C 180,E1 -28190.563,E2 -28190.563} C_VEL
LIN {X 0,Y 83.021,Z 579.976,A -85,B 0,C 180,E1 -28200.527,E2 -28200.527} C_VEL
LIN {X 0,Y 88.733,Z 585.048,A -85,B 0,C 180,E1 -28209.32,E2 -28209.32} C_VEL
LIN {X 0,Y 94.362,Z 588.182,A -85,B 0,C 180,E1 -28214.869,E2 -28214.869} C_VEL
LIN {X 0,Y 95.414,Z 588.508,A -85,B 0,C 180,E1 -28217.007,E2 -28217.007} C_VEL
LIN {X 0,Y 86.325,Z 580.9,A -85,B 0,C 180,E1 -28225.259,E2 -28225.259} C_VEL
LIN {X 0,Y 80.38,Z 572.891,A -85,B 0,C 180,E1 -28234.078,E2 -28234.078} C_VEL
LIN {X 0,Y 77.272,Z 564.824,A -85,B 0,C 180,E1 -28242.808,E2 -28242.808} C_VEL
LIN {X 0,Y 75.776,Z 556.396,A -85,B 0,C 180,E1 -28250.66,E2 -28250.66} C_VEL
LIN {X 0,Y 75.03,Z 546.228,A -85,B 0,C 180,E1 -28258.659,E2 -28258.659} C_VEL
LIN {X 0,Y 75.144,Z 534.47,A -85,B 0,C 180,E1 -28266.041,E2 -28266.041} C_VEL
LIN {X 0,Y 75.879,Z 522.75,A -85,B 0,C 180,E1 -28272.03,E2 -28272.03} C_VEL
LIN {X 0,Y 75.917,Z 520.397,A -85,B 0,C 180,E1 -28273.042,E2 -28273.042} C_VEL
LIN {X 0,Y 72.962,Z 507.394,A -85,B 0,C 180,E1 -28277.159,E2 -28277.159} C_VEL
LIN {X 0,Y 71.606,Z 507.565,A -85,B 0,C 180,E1 -28289.391,E2 -28289.391} C_VEL
LIN {X 0,Y 72.056,Z 507.508,A -85,B 0,C 180,E1 -28298.712,E2 -28298.712} C_VEL
LIN {X 0,Y 72.216,Z 507.489,A -85,B 0,C 180,E1 -28307.058,E2 -28307.058} C_VEL
LIN {X 0,Y 72.303,Z 507.479,A -85,B 0,C 180,E1 -28314.322,E2 -28314.322} C_VEL
LIN {X 0,Y 72.378,Z 507.463,A -85,B 0,C 180,E1 -28320.953,E2 -28320.953} C_VEL
LIN {X 0,Y 72.397,Z 507.459,A -85,B 0,C 180,E1 -28327.15,E2 -28327.15} C_VEL
LIN {X 0,Y 72.725,Z 507.421,A -85,B 0,C 180,E1 -28335.109,E2 -28335.109} C_VEL
LIN {X 0,Y 72.838,Z 507.398,A -85,B 0,C 180,E1 -28340.468,E2 -28340.468} C_VEL
LIN {X 0,Y 73.573,Z 507.321,A -85,B 0,C 180,E1 -28349.999,E2 -28349.999} C_VEL
LIN {X 0,Y 72.861,Z 507.405,A -85,B 0,C 180,E1 -28361.122,E2 -28361.122} C_VEL
LIN {X 0,Y 72.728,Z 507.417,A -85,B 0,C 180,E1 -28363.957,E2 -28363.957} C_VEL
LIN {X 0,Y 72.325,Z 507.476,A -85,B 0,C 180,E1 -28367.035,E2 -28367.035} C_VEL
LIN {X 0,Y 70.777,Z 507.674,A -85,B 0,C 180,E1 -28371.608,E2 -28371.608} C_VEL
LIN {X 0,Y 67.274,Z 508.103,A -85,B 0,C 180,E1 -28379.465,E2 -28379.465} C_VEL
LIN {X 0,Y 65.16,Z 508.361,A -85,B 0,C 180,E1 -28388.15,E2 -28388.15} C_VEL
LIN {X 0,Y 65.187,Z 508.353,A -85,B 0,C 180,E1 -28389.949,E2 -28389.949} C_VEL
LIN {X 0,Y 65.208,Z 508.355,A -85,B 0,C 180,E1 -28399.707,E2 -28399.707} C_VEL
LIN {X 0,Y 65.254,Z 508.354,A -85,B 0,C 180,E1 -28409.497,E2 -28409.497} C_VEL
LIN {X 0,Y 65.241,Z 508.351,A -85,B 0,C 180,E1 -28414.474,E2 -28414.474} C_VEL
LIN {X 0,Y 65.651,Z 508.297,A -85,B 0,C 180,E1 -28424.457,E2 -28424.457} C_VEL
LIN {X 0,Y 65.783,Z 508.289,A -85,B 0,C 180,E1 -28427.661,E2 -28427.661} C_VEL
LIN {X 0,Y 66.505,Z 508.197,A -85,B 0,C 180,E1 -28439.999,E2 -28439.999} C_VEL
LIN {X 0,Y 65.775,Z 508.285,A -85,B 0,C 180,E1 -28452.338,E2 -28452.338} C_VEL
LIN {X 0,Y 65.385,Z 508.332,A -85,B 0,C 180,E1 -28458.81,E2 -28458.81} C_VEL
LIN {X 0,Y 65.246,Z 508.356,A -85,B 0,C 180,E1 -28465.521,E2 -28465.521} C_VEL
LIN {X 0,Y 65.247,Z 508.358,A -85,B 0,C 180,E1 -28472.585,E2 -28472.585} C_VEL
LIN {X 0,Y 65.527,Z 508.323,A -85,B 0,C 180,E1 -28481.344,E2 -28481.344} C_VEL
LIN {X 0,Y 65.814,Z 508.288,A -85,B 0,C 180,E1 -28490.157,E2 -28490.157} C_VEL
LIN {X 0,Y 64.726,Z 508.419,A -85,B 0,C 180,E1 -28500.299,E2 -28500.299} C_VEL
LIN {X 0,Y 65.255,Z 508.364,A -85,B 0,C 180,E1 -28512.455,E2 -28512.455} C_VEL
LIN {X 0,Y 66.741,Z 523.338,A -85,B 0,C 180,E1 -28517.844,E2 -28517.844} C_VEL
LIN {X 0,Y 69.403,Z 536.635,A -85,B 0,C 180,E1 -28523.46,E2 -28523.46} C_VEL
LIN {X 0,Y 71.57,Z 544.557,A -85,B 0,C 180,E1 -28527.187,E2 -28527.187} C_VEL
LIN {X 0,Y 72.518,Z 554.759,A -85,B 0,C 180,E1 -28534.392,E2 -28534.392} C_VEL
LIN {X 0,Y 73.641,Z 560.931,A -85,B 0,C 180,E1 -28539.571,E2 -28539.571} C_VEL
LIN {X 0,Y 73.903,Z 562.348,A -85,B 0,C 180,E1 -28540.965,E2 -28540.965} C_VEL
LIN {X 0,Y 74.167,Z 568.965,A -85,B 0,C 180,E1 -28550.199,E2 -28550.199} C_VEL
LIN {X 0,Y 77.795,Z 576.451,A -85,B 0,C 180,E1 -28562.824,E2 -28562.824} C_VEL
LIN {X 0,Y 83.961,Z 581.757,A -85,B 0,C 180,E1 -28572.041,E2 -28572.041} C_VEL
LIN {X 0,Y 87.91,Z 584.124,A -85,B 0,C 180,E1 -28576.016,E2 -28576.016} C_VEL
LIN {X 0,Y 81.042,Z 578.011,A -85,B 0,C 180,E1 -28582.625,E2 -28582.625} C_VEL
LIN {X 0,Y 74.685,Z 569.653,A -85,B 0,C 180,E1 -28591.934,E2 -28591.934} C_VEL
LIN {X 0,Y 71.295,Z 561.114,A -85,B 0,C 180,E1 -28601.316,E2 -28601.316} C_VEL
LIN {X 0,Y 69.566,Z 552.247,A -85,B 0,C 180,E1 -28609.818,E2 -28609.818} C_VEL
LIN {X 0,Y 68.822,Z 543.258,A -85,B 0,C 180,E1 -28617.075,E2 -28617.075} C_VEL
LIN {X 0,Y 68.666,Z 532.448,A -85,B 0,C 180,E1 -28624.404,E2 -28624.404} C_VEL
LIN {X 0,Y 69.26,Z 520.296,A -85,B 0,C 180,E1 -28630.97,E2 -28630.97} C_VEL
LIN {X 0,Y 66.315,Z 508.218,A -85,B 0,C 180,E1 -28635.247,E2 -28635.247} C_VEL
LIN {X 0,Y 64.592,Z 508.434,A -85,B 0,C 180,E1 -28645.801,E2 -28645.801} C_VEL
LIN {X 0,Y 64.629,Z 508.425,A -85,B 0,C 180,E1 -28652.939,E2 -28652.939} C_VEL
LIN {X 0,Y 64.997,Z 508.38,A -85,B 0,C 180,E1 -28660.806,E2 -28660.806} C_VEL
LIN {X 0,Y 65.19,Z 508.356,A -85,B 0,C 180,E1 -28669.694,E2 -28669.694} C_VEL
LIN {X 0,Y 65.258,Z 508.346,A -85,B 0,C 180,E1 -28679.497,E2 -28679.497} C_VEL
LIN {X 0,Y 65.242,Z 508.358,A -85,B 0,C 180,E1 -28684.475,E2 -28684.475} C_VEL
LIN {X 0,Y 65.628,Z 508.307,A -85,B 0,C 180,E1 -28694.542,E2 -28694.542} C_VEL
LIN {X 0,Y 65.758,Z 508.285,A -85,B 0,C 180,E1 -28697.656,E2 -28697.656} C_VEL
LIN {X 0,Y 66.496,Z 508.203,A -85,B 0,C 180,E1 -28709.999,E2 -28709.999} C_VEL
LIN {X 0,Y 65.757,Z 508.285,A -85,B 0,C 180,E1 -28722.341,E2 -28722.341} C_VEL
LIN {X 0,Y 65.382,Z 508.34,A -85,B 0,C 180,E1 -28728.811,E2 -28728.811} C_VEL
LIN {X 0,Y 65.241,Z 508.358,A -85,B 0,C 180,E1 -28735.523,E2 -28735.523} C_VEL
LIN {X 0,Y 65.199,Z 508.358,A -85,B 0,C 180,E1 -28742.611,E2 -28742.611} C_VEL
LIN {X 0,Y 65.187,Z 508.353,A -85,B 0,C 180,E1 -28749.949,E2 -28749.949} C_VEL
LIN {X 0,Y 65.036,Z 508.397,A -85,B 0,C 180,E1 -28753.381,E2 -28753.381} C_VEL
LIN {X 0,Y 63.756,Z 508.581,A -85,B 0,C 180,E1 -28758.509,E2 -28758.509} C_VEL
LIN {X 0,Y 61.841,Z 508.828,A -85,B 0,C 180,E1 -28763.673,E2 -28763.673} C_VEL
LIN {X 0,Y 58.438,Z 509.222,A -85,B 0,C 180,E1 -28775.141,E2 -28775.141} C_VEL
LIN {X 0,Y 58.206,Z 509.23,A -85,B 0,C 180,E1 -28779.216,E2 -28779.216} C_VEL
LIN {X 0,Y 58.659,Z 509.17,A -85,B 0,C 180,E1 -28786.134,E2 -28786.134} C_VEL
LIN {X 0,Y 58.824,Z 509.148,A -85,B 0,C 180,E1 -28793.137,E2 -28793.137} C_VEL
LIN {X 0,Y 59.397,Z 509.082,A -85,B 0,C 180,E1 -28799.998,E2 -28799.998} C_VEL
LIN {X 0,Y 58.823,Z 509.158,A -85,B 0,C 180,E1 -28806.86,E2 -28806.86} C_VEL
LIN {X 0,Y 58.525,Z 509.195,A -85,B 0,C 180,E1 -28816.124,E2 -28816.124} C_VEL
LIN {X 0,Y 58.169,Z 509.229,A -85,B 0,C 180,E1 -28828.898,E2 -28828.898} C_VEL
LIN {X 0,Y 58.197,Z 509.226,A -85,B 0,C 180,E1 -28837.142,E2 -28837.142} C_VEL
LIN {X 0,Y 58.552,Z 509.183,A -85,B 0,C 180,E1 -28846.067,E2 -28846.067} C_VEL
LIN {X 0,Y 58.291,Z 509.221,A -85,B 0,C 180,E1 -28852.929,E2 -28852.929} C_VEL
LIN {X 0,Y 57.611,Z 509.306,A -85,B 0,C 180,E1 -28860.795,E2 -28860.795} C_VEL
LIN {X 0,Y 58.677,Z 509.173,A -85,B 0,C 180,E1 -28875.099,E2 -28875.099} C_VEL
LIN {X 0,Y 60.655,Z 524.349,A -85,B 0,C 180,E1 -28881.254,E2 -28881.254} C_VEL
LIN {X 0,Y 63.992,Z 538.361,A -85,B 0,C 180,E1 -28887.766,E2 -28887.766} C_VEL
LIN {X 0,Y 65.404,Z 542.792,A -85,B 0,C 180,E1 -28890.001,E2 -28890.001} C_VEL
LIN {X 0,Y 66.561,Z 550.911,A -85,B 0,C 180,E1 -28896.062,E2 -28896.062} C_VEL
LIN {X 0,Y 68.004,Z 557.699,A -85,B 0,C 180,E1 -28901.93,E2 -28901.93} C_VEL
LIN {X 0,Y 68.285,Z 559.494,A -85,B 0,C 180,E1 -28903.888,E2 -28903.888} C_VEL
LIN {X 0,Y 69.097,Z 566.16,A -85,B 0,C 180,E1 -28914.008,E2 -28914.008} C_VEL
LIN {X 0,Y 72.795,Z 572.733,A -85,B 0,C 180,E1 -28925.401,E2 -28925.401} C_VEL
LIN {X 0,Y 79.487,Z 578.295,A -85,B 0,C 180,E1 -28935.02,E2 -28935.02} C_VEL
LIN {X 0,Y 78.082,Z 576.934,A -85,B 0,C 180,E1 -28937.561,E2 -28937.561} C_VEL
LIN {X 0,Y 69.217,Z 566.129,A -85,B 0,C 180,E1 -28949.492,E2 -28949.492} C_VEL
LIN {X 0,Y 65.936,Z 558.522,A -85,B 0,C 180,E1 -28958.097,E2 -28958.097} C_VEL
LIN {X 0,Y 63.757,Z 549.462,A -85,B 0,C 180,E1 -28967.265,E2 -28967.265} C_VEL
LIN {X 0,Y 62.691,Z 540.127,A -85,B 0,C 180,E1 -28975.178,E2 -28975.178} C_VEL
LIN {X 0,Y 62.39,Z 528.744,A -85,B 0,C 180,E1 -28983.23,E2 -28983.23} C_VEL
LIN {X 0,Y 62.64,Z 520.642,A -85,B 0,C 180,E1 -28988.064,E2 -28988.064} C_VEL
LIN {X 0,Y 62.179,Z 517.757,A -85,B 0,C 180,E1 -28989.352,E2 -28989.352} C_VEL
LIN {X 0,Y 59.948,Z 509.017,A -85,B 0,C 180,E1 -28992.485,E2 -28992.485} C_VEL
LIN {X 0,Y 57.85,Z 509.277,A -85,B 0,C 180,E1 -29001.376,E2 -29001.376} C_VEL
LIN {X 0,Y 57.54,Z 509.311,A -85,B 0,C 180,E1 -29011.239,E2 -29011.239} C_VEL
LIN {X 0,Y 57.686,Z 509.3,A -85,B 0,C 180,E1 -29017.531,E2 -29017.531} C_VEL
LIN {X 0,Y 57.889,Z 509.267,A -85,B 0,C 180,E1 -29023.242,E2 -29023.242} C_VEL
LIN {X 0,Y 57.955,Z 509.266,A -85,B 0,C 180,E1 -29026.688,E2 -29026.688} C_VEL
LIN {X 0,Y 58.026,Z 509.252,A -85,B 0,C 180,E1 -29032.727,E2 -29032.727} C_VEL
LIN {X 0,Y 58.162,Z 509.232,A -85,B 0,C 180,E1 -29037.766,E2 -29037.766} C_VEL
LIN {X 0,Y 58.154,Z 509.235,A -85,B 0,C 180,E1 -29041.09,E2 -29041.09} C_VEL
LIN {X 0,Y 58.52,Z 509.193,A -85,B 0,C 180,E1 -29053.906,E2 -29053.906} C_VEL
LIN {X 0,Y 58.803,Z 509.157,A -85,B 0,C 180,E1 -29063.134,E2 -29063.134} C_VEL
LIN {X 0,Y 59.386,Z 509.088,A -85,B 0,C 180,E1 -29069.999,E2 -29069.999} C_VEL
LIN {X 0,Y 58.801,Z 509.157,A -85,B 0,C 180,E1 -29076.863,E2 -29076.863} C_VEL
LIN {X 0,Y 58.519,Z 509.194,A -85,B 0,C 180,E1 -29086.092,E2 -29086.092} C_VEL
LIN {X 0,Y 58.153,Z 509.235,A -85,B 0,C 180,E1 -29098.907,E2 -29098.907} C_VEL
LIN {X 0,Y 58.161,Z 509.233,A -85,B 0,C 180,E1 -29102.232,E2 -29102.232} C_VEL
LIN {X 0,Y 57.95,Z 509.254,A -85,B 0,C 180,E1 -29109.881,E2 -29109.881} C_VEL
LIN {X 0,Y 58.019,Z 509.251,A -85,B 0,C 180,E1 -29116.616,E2 -29116.616} C_VEL
LIN {X 0,Y 58.035,Z 509.256,A -85,B 0,C 180,E1 -29122.733,E2 -29122.733} C_VEL
LIN {X 0,Y 58.157,Z 509.231,A -85,B 0,C 180,E1 -29127.767,E2 -29127.767} C_VEL
LIN {X 0,Y 58.152,Z 509.241,A -85,B 0,C 180,E1 -29131.089,E2 -29131.089} C_VEL
LIN {X 0,Y 58.206,Z 509.23,A -85,B 0,C 180,E1 -29139.216,E2 -29139.216} C_VEL
LIN {X 0,Y 57.795,Z 509.279,A -85,B 0,C 180,E1 -29143.069,E2 -29143.069} C_VEL
LIN {X 0,Y 56.652,Z 509.423,A -85,B 0,C 180,E1 -29146.875,E2 -29146.875} C_VEL
LIN {X 0,Y 52.206,Z 509.973,A -85,B 0,C 180,E1 -29160.567,E2 -29160.567} C_VEL
LIN {X 0,Y 51.697,Z 510.044,A -85,B 0,C 180,E1 -29167.812,E2 -29167.812} C_VEL
LIN {X 0,Y 51.393,Z 510.081,A -85,B 0,C 180,E1 -29176.818,E2 -29176.818} C_VEL
LIN {X 0,Y 51.033,Z 510.128,A -85,B 0,C 180,E1 -29184.401,E2 -29184.401} C_VEL
LIN {X 0,Y 51.112,Z 510.116,A -85,B 0,C 180,E1 -29194.414,E2 -29194.414} C_VEL
LIN {X 0,Y 51.357,Z 510.086,A -85,B 0,C 180,E1 -29203.173,E2 -29203.173} C_VEL
LIN {X 0,Y 51.42,Z 510.071,A -85,B 0,C 180,E1 -29206.893,E2 -29206.893} C_VEL
LIN {X 0,Y 50.875,Z 510.142,A -85,B 0,C 180,E1 -29216.458,E2 -29216.458} C_VEL
LIN {X 0,Y 52.225,Z 509.974,A -85,B 0,C 180,E1 -29238.356,E2 -29238.356} C_VEL
LIN {X 0,Y 52.46,Z 510.214,A -85,B 0,C 180,E1 -29238.898,E2 -29238.898} C_VEL
LIN {X 0,Y 54.632,Z 523.795,A -85,B 0,C 180,E1 -29244.937,E2 -29244.937} C_VEL
LIN {X 0,Y 58.359,Z 537.467,A -85,B 0,C 180,E1 -29251.727,E2 -29251.727} C_VEL
LIN {X 0,Y 59.941,Z 542.073,A -85,B 0,C 180,E1 -29254.204,E2 -29254.204} C_VEL
LIN {X 0,Y 61.587,Z 550.889,A -85,B 0,C 180,E1 -29261.521,E2 -29261.521} C_VEL
LIN {X 0,Y 62.817,Z 555.76,A -85,B 0,C 180,E1 -29266.217,E2 -29266.217} C_VEL
LIN {X 0,Y 64.268,Z 562.913,A -85,B 0,C 180,E1 -29277.873,E2 -29277.873} C_VEL
LIN {X 0,Y 68.096,Z 568.731,A -85,B 0,C 180,E1 -29288.263,E2 -29288.263} C_VEL
LIN {X 0,Y 71.404,Z 571.782,A -85,B 0,C 180,E1 -29293.551,E2 -29293.551} C_VEL
LIN {X 0,Y 71.951,Z 572.104,A -85,B 0,C 180,E1 -29295.747,E2 -29295.747} C_VEL
LIN {X 0,Y 64.039,Z 562.3,A -85,B 0,C 180,E1 -29306.722,E2 -29306.722} C_VEL
LIN {X 0,Y 60.319,Z 554.342,A -85,B 0,C 180,E1 -29315.935,E2 -29315.935} C_VEL
LIN {X 0,Y 58.207,Z 546.39,A -85,B 0,C 180,E1 -29324.238,E2 -29324.238} C_VEL
LIN {X 0,Y 56.727,Z 536.793,A -85,B 0,C 180,E1 -29332.885,E2 -29332.885} C_VEL
LIN {X 0,Y 56.208,Z 527.453,A -85,B 0,C 180,E1 -29340.002,E2 -29340.002} C_VEL
LIN {X 0,Y 56.258,Z 519.191,A -85,B 0,C 180,E1 -29345.378,E2 -29345.378} C_VEL
LIN {X 0,Y 53.678,Z 509.798,A -85,B 0,C 180,E1 -29349.184,E2 -29349.184} C_VEL
LIN {X 0,Y 51.399,Z 510.076,A -85,B 0,C 180,E1 -29356.831,E2 -29356.831} C_VEL
LIN {X 0,Y 50.493,Z 510.186,A -85,B 0,C 180,E1 -29373.834,E2 -29373.834} C_VEL
LIN {X 0,Y 50.841,Z 510.146,A -85,B 0,C 180,E1 -29383.726,E2 -29383.726} C_VEL
LIN {X 0,Y 50.907,Z 510.144,A -85,B 0,C 180,E1 -29386.345,E2 -29386.345} C_VEL
LIN {X 0,Y 51.051,Z 510.122,A -85,B 0,C 180,E1 -29396.585,E2 -29396.585} C_VEL
LIN {X 0,Y 51.026,Z 510.125,A -85,B 0,C 180,E1 -29405.592,E2 -29405.592} C_VEL
LIN {X 0,Y 51.461,Z 510.072,A -85,B 0,C 180,E1 -29414.147,E2 -29414.147} C_VEL
LIN {X 0,Y 51.68,Z 510.047,A -85,B 0,C 180,E1 -29422.182,E2 -29422.182} C_VEL
LIN {X 0,Y 52.27,Z 509.975,A -85,B 0,C 180,E1 -29429.998,E2 -29429.998} C_VEL
LIN {X 0,Y 51.678,Z 510.047,A -85,B 0,C 180,E1 -29437.814,E2 -29437.814} C_VEL
LIN {X 0,Y 51.388,Z 510.084,A -85,B 0,C 180,E1 -29446.789,E2 -29446.789} C_VEL
LIN {X 0,Y 51.025,Z 510.125,A -85,B 0,C 180,E1 -29454.405,E2 -29454.405} C_VEL
LIN {X 0,Y 51.033,Z 510.127,A -85,B 0,C 180,E1 -29464.277,E2 -29464.277} C_VEL
LIN {X 0,Y 50.986,Z 510.127,A -85,B 0,C 180,E1 -29476.43,E2 -29476.43} C_VEL
LIN {X 0,Y 51.05,Z 510.116,A -85,B 0,C 180,E1 -29486.584,E2 -29486.584} C_VEL
LIN {X 0,Y 51.026,Z 510.119,A -85,B 0,C 180,E1 -29495.592,E2 -29495.592} C_VEL
LIN {X 0,Y 51.482,Z 510.062,A -85,B 0,C 180,E1 -29504.153,E2 -29504.153} C_VEL
LIN {X 0,Y 51.7,Z 510.036,A -85,B 0,C 180,E1 -29512.185,E2 -29512.185} C_VEL
LIN {X 0,Y 52.206,Z 509.973,A -85,B 0,C 180,E1 -29520.567,E2 -29520.567} C_VEL
LIN {X 0,Y 50.881,Z 510.147,A -85,B 0,C 180,E1 -29526.969,E2 -29526.969} C_VEL
LIN {X 0,Y 48.939,Z 510.384,A -85,B 0,C 180,E1 -29533.434,E2 -29533.434} C_VEL
LIN {X 0,Y 45.035,Z 510.866,A -85,B 0,C 180,E1 -29547.552,E2 -29547.552} C_VEL
LIN {X 0,Y 44.037,Z 510.99,A -85,B 0,C 180,E1 -29558.042,E2 -29558.042} C_VEL
LIN {X 0,Y 44.013,Z 511.003,A -85,B 0,C 180,E1 -29570.307,E2 -29570.307} C_VEL
LIN {X 0,Y 43.472,Z 511.066,A -85,B 0,C 180,E1 -29580.99,E2 -29580.99} C_VEL
LIN {X 0,Y 45.954,Z 510.754,A -85,B 0,C 180,E1 -29602.312,E2 -29602.312} C_VEL
LIN {X 0,Y 46.452,Z 510.745,A -85,B 0,C 180,E1 -29603.486,E2 -29603.486} C_VEL
LIN {X 0,Y 49.195,Z 524.303,A -85,B 0,C 180,E1 -29610.092,E2 -29610.092} C_VEL
LIN {X 0,Y 53.825,Z 538.505,A -85,B 0,C 180,E1 -29617.504,E2 -29617.504} C_VEL
LIN {X 0,Y 54.702,Z 541.184,A -85,B 0,C 180,E1 -29619.243,E2 -29619.243} C_VEL
LIN {X 0,Y 57.279,Z 550.65,A -85,B 0,C 180,E1 -29627.865,E2 -29627.865} C_VEL
LIN {X 0,Y 57.752,Z 552.172,A -85,B 0,C 180,E1 -29629.553,E2 -29629.553} C_VEL
LIN {X 0,Y 59.847,Z 559.588,A -85,B 0,C 180,E1 -29642.299,E2 -29642.299} C_VEL
LIN {X 0,Y 63.699,Z 564.561,A -85,B 0,C 180,E1 -29651.454,E2 -29651.454} C_VEL
LIN {X 0,Y 64.761,Z 565.513,A -85,B 0,C 180,E1 -29655.14,E2 -29655.14} C_VEL
LIN {X 0,Y 57.601,Z 555.553,A -85,B 0,C 180,E1 -29666.7,E2 -29666.7} C_VEL
LIN {X 0,Y 53.853,Z 546.645,A -85,B 0,C 180,E1 -29676.953,E2 -29676.953} C_VEL
LIN {X 0,Y 51.702,Z 537.372,A -85,B 0,C 180,E1 -29686.24,E2 -29686.24} C_VEL
LIN {X 0,Y 50.413,Z 527.158,A -85,B 0,C 180,E1 -29695.003,E2 -29695.003} C_VEL
LIN {X 0,Y 50.045,Z 518.008,A -85,B 0,C 180,E1 -29701.814,E2 -29701.814} C_VEL
LIN {X 0,Y 47.691,Z 510.54,A -85,B 0,C 180,E1 -29704.969,E2 -29704.969} C_VEL
LIN {X 0,Y 46.084,Z 510.741,A -85,B 0,C 180,E1 -29708.774,E2 -29708.774} C_VEL
LIN {X 0,Y 43.351,Z 511.085,A -85,B 0,C 180,E1 -29729.104,E2 -29729.104} C_VEL
LIN {X 0,Y 43.491,Z 511.059,A -85,B 0,C 180,E1 -29740.273,E2 -29740.273} C_VEL
LIN {X 0,Y 43.762,Z 511.023,A -85,B 0,C 180,E1 -29750.028,E2 -29750.028} C_VEL
LIN {X 0,Y 43.827,Z 511.022,A -85,B 0,C 180,E1 -29753.305,E2 -29753.305} C_VEL
LIN {X 0,Y 43.844,Z 511.016,A -85,B 0,C 180,E1 -29761.255,E2 -29761.255} C_VEL
LIN {X 0,Y 44.231,Z 510.976,A -85,B 0,C 180,E1 -29772.439,E2 -29772.439} C_VEL
LIN {X 0,Y 44.533,Z 510.938,A -85,B 0,C 180,E1 -29780.918,E2 -29780.918} C_VEL
LIN {X 0,Y 45.144,Z 510.862,A -85,B 0,C 180,E1 -29789.998,E2 -29789.998} C_VEL
LIN {X 0,Y 44.531,Z 510.938,A -85,B 0,C 180,E1 -29799.078,E2 -29799.078} C_VEL
LIN {X 0,Y 44.155,Z 510.983,A -85,B 0,C 180,E1 -29808.56,E2 -29808.56} C_VEL
LIN {X 0,Y 43.845,Z 511.016,A -85,B 0,C 180,E1 -29818.74,E2 -29818.74} C_VEL
LIN {X 0,Y 43.807,Z 511.018,A -85,B 0,C 180,E1 -29829.918,E2 -29829.918} C_VEL
LIN {X 0,Y 43.843,Z 511.023,A -85,B 0,C 180,E1 -29843.27,E2 -29843.27} C_VEL
LIN {X 0,Y 43.844,Z 511.024,A -85,B 0,C 180,E1 -29851.254,E2 -29851.254} C_VEL
LIN {X 0,Y 44.257,Z 510.966,A -85,B 0,C 180,E1 -29862.318,E2 -29862.318} C_VEL
LIN {X 0,Y 44.552,Z 510.93,A -85,B 0,C 180,E1 -29870.922,E2 -29870.922} C_VEL
LIN {X 0,Y 45.156,Z 510.854,A -85,B 0,C 180,E1 -29879.998,E2 -29879.998} C_VEL
LIN {X 0,Y 44.546,Z 510.929,A -85,B 0,C 180,E1 -29889.075,E2 -29889.075} C_VEL
LIN {X 0,Y 44.157,Z 510.975,A -85,B 0,C 180,E1 -29898.559,E2 -29898.559} C_VEL
LIN {X 0,Y 43.887,Z 511.008,A -85,B 0,C 180,E1 -29908.71,E2 -29908.71} C_VEL
LIN {X 0,Y 44.037,Z 510.99,A -85,B 0,C 180,E1 -29918.042,E2 -29918.042} C_VEL
LIN {X 0,Y 43.661,Z 511.044,A -85,B 0,C 180,E1 -29923.067,E2 -29923.067} C_VEL
LIN {X 0,Y 42.015,Z 511.254,A -85,B 0,C 180,E1 -29930.609,E2 -29930.609} C_VEL
LIN {X 0,Y 38.601,Z 511.671,A -85,B 0,C 180,E1 -29944.238,E2 -29944.238} C_VEL
LIN {X 0,Y 37.652,Z 511.794,A -85,B 0,C 180,E1 -29956.69,E2 -29956.69} C_VEL
LIN {X 0,Y 38.546,Z 511.674,A -85,B 0,C 180,E1 -29962.762,E2 -29962.762} C_VEL
LIN {X 0,Y 40.915,Z 511.38,A -85,B 0,C 180,E1 -29969.541,E2 -29969.541} C_VEL
LIN {X 0,Y 44.628,Z 525.599,A -85,B 0,C 180,E1 -29977.007,E2 -29977.007} C_VEL
LIN {X 0,Y 49.203,Z 537.579,A -85,B 0,C 180,E1 -29983.423,E2 -29983.423} C_VEL
LIN {X 0,Y 50.043,Z 539.984,A -85,B 0,C 180,E1 -29985.269,E2 -29985.269} C_VEL
LIN {X 0,Y 52.319,Z 546.775,A -85,B 0,C 180,E1 -29991.681,E2 -29991.681} C_VEL
LIN {X 0,Y 52.969,Z 548.423,A -85,B 0,C 180,E1 -29993.458,E2 -29993.458} C_VEL
LIN {X 0,Y 54.767,Z 553.914,A -85,B 0,C 180,E1 -30003.273,E2 -30003.273} C_VEL
LIN {X 0,Y 57.929,Z 558.445,A -85,B 0,C 180,E1 -30011.863,E2 -30011.863} C_VEL
LIN {X 0,Y 58.436,Z 558.98,A -85,B 0,C 180,E1 -30013.814,E2 -30013.814} C_VEL
LIN {X 0,Y 52.217,Z 549.923,A -85,B 0,C 180,E1 -30024.579,E2 -30024.579} C_VEL
LIN {X 0,Y 48.569,Z 541.472,A -85,B 0,C 180,E1 -30034.274,E2 -30034.274} C_VEL
LIN {X 0,Y 46.148,Z 532.545,A -85,B 0,C 180,E1 -30043.41,E2 -30043.41} C_VEL
LIN {X 0,Y 44.585,Z 521.46,A -85,B 0,C 180,E1 -30053.212,E2 -30053.212} C_VEL
LIN {X 0,Y 44.304,Z 517.237,A -85,B 0,C 180,E1 -30056.592,E2 -30056.592} C_VEL
LIN {X 0,Y 42.317,Z 511.208,A -85,B 0,C 180,E1 -30059.093,E2 -30059.093} C_VEL
LIN {X 0,Y 38.15,Z 511.733,A -85,B 0,C 180,E1 -30070.618,E2 -30070.618} C_VEL
LIN {X 0,Y 36.332,Z 511.953,A -85,B 0,C 180,E1 -30095.476,E2 -30095.476} C_VEL
LIN {X 0,Y 36.421,Z 511.941,A -85,B 0,C 180,E1 -30099.474,E2 -30099.474} C_VEL
LIN {X 0,Y 36.68,Z 511.905,A -85,B 0,C 180,E1 -30110.038,E2 -30110.038} C_VEL
LIN {X 0,Y 36.713,Z 511.912,A -85,B 0,C 180,E1 -30114.947,E2 -30114.947} C_VEL
LIN {X 0,Y 37.058,Z 511.866,A -85,B 0,C 180,E1 -30131.495,E2 -30131.495} C_VEL
LIN {X 0,Y 37.33,Z 511.828,A -85,B 0,C 180,E1 -30139.146,E2 -30139.146} C_VEL
LIN {X 0,Y 38.002,Z 511.752,A -85,B 0,C 180,E1 -30149.998,E2 -30149.998} C_VEL
LIN {X 0,Y 37.329,Z 511.828,A -85,B 0,C 180,E1 -30160.85,E2 -30160.85} C_VEL
LIN {X 0,Y 37.057,Z 511.867,A -85,B 0,C 180,E1 -30168.5,E2 -30168.5} C_VEL
LIN {X 0,Y 36.726,Z 511.911,A -85,B 0,C 180,E1 -30185.033,E2 -30185.033} C_VEL
LIN {X 0,Y 36.727,Z 511.9,A -85,B 0,C 180,E1 -30190.05,E2 -30190.05} C_VEL
LIN {X 0,Y 36.726,Z 511.901,A -85,B 0,C 180,E1 -30199.944,E2 -30199.944} C_VEL
LIN {X 0,Y 36.722,Z 511.903,A -85,B 0,C 180,E1 -30204.957,E2 -30204.957} C_VEL
LIN {X 0,Y 37.08,Z 511.863,A -85,B 0,C 180,E1 -30221.379,E2 -30221.379} C_VEL
LIN {X 0,Y 37.349,Z 511.833,A -85,B 0,C 180,E1 -30229.151,E2 -30229.151} C_VEL
LIN {X 0,Y 38.015,Z 511.742,A -85,B 0,C 180,E1 -30239.997,E2 -30239.997} C_VEL
LIN {X 0,Y 37.338,Z 511.823,A -85,B 0,C 180,E1 -30250.847,E2 -30250.847} C_VEL
LIN {X 0,Y 37.061,Z 511.859,A -85,B 0,C 180,E1 -30258.536,E2 -30258.536} C_VEL
LIN {X 0,Y 36.849,Z 511.888,A -85,B 0,C 180,E1 -30274.899,E2 -30274.899} C_VEL
LIN {X 0,Y 36.955,Z 511.878,A -85,B 0,C 180,E1 -30280.476,E2 -30280.476} C_VEL
LIN {X 0,Y 36.917,Z 511.884,A -85,B 0,C 180,E1 -30289.592,E2 -30289.592} C_VEL
LIN {X 0,Y 36.64,Z 511.91,A -85,B 0,C 180,E1 -30294.873,E2 -30294.873} C_VEL
LIN {X 0,Y 38.546,Z 511.674,A -85,B 0,C 180,E1 -30322.762,E2 -30322.762} C_VEL
LIN {X 0,Y 39.152,Z 512.075,A -85,B 0,C 180,E1 -30326.657,E2 -30326.657} C_VEL
LIN {X 0,Y 39.231,Z 513.711,A -85,B 0,C 180,E1 -30331.587,E2 -30331.587} C_VEL
LIN {X 0,Y 38.923,Z 516.916,A -85,B 0,C 180,E1 -30337.171,E2 -30337.171} C_VEL
LIN {X 0,Y 39.004,Z 520.059,A -85,B 0,C 180,E1 -30340.892,E2 -30340.892} C_VEL
LIN {X 0,Y 39.836,Z 523.884,A -85,B 0,C 180,E1 -30343.953,E2 -30343.953} C_VEL
LIN {X 0,Y 41.237,Z 527.813,A -85,B 0,C 180,E1 -30346.242,E2 -30346.242} C_VEL
LIN {X 0,Y 44.717,Z 535.436,A -85,B 0,C 180,E1 -30349.94,E2 -30349.94} C_VEL
LIN {X 0,Y 45.953,Z 538.344,A -85,B 0,C 180,E1 -30352.008,E2 -30352.008} C_VEL
LIN {X 0,Y 48.6,Z 544.749,A -85,B 0,C 180,E1 -30358.328,E2 -30358.328} C_VEL
LIN {X 0,Y 52.406,Z 551.876,A -85,B 0,C 180,E1 -30372.111,E2 -30372.111} C_VEL
LIN {X 0,Y 48.802,Z 546.902,A -85,B 0,C 180,E1 -30378.375,E2 -30378.375} C_VEL
LIN {X 0,Y 44.226,Z 537.738,A -85,B 0,C 180,E1 -30388.907,E2 -30388.907} C_VEL
LIN {X 0,Y 41.167,Z 528.409,A -85,B 0,C 180,E1 -30398.741,E2 -30398.741} C_VEL
LIN {X 0,Y 39.204,Z 518.16,A -85,B 0,C 180,E1 -30408.368,E2 -30408.368} C_VEL
LIN {X 0,Y 39.058,Z 516.728,A -85,B 0,C 180,E1 -30409.636,E2 -30409.636} C_VEL
LIN {X 0,Y 37.341,Z 511.829,A -85,B 0,C 180,E1 -30411.838,E2 -30411.838} C_VEL
LIN {X 0,Y 33.566,Z 512.288,A -85,B 0,C 180,E1 -30420.003,E2 -30420.003} C_VEL
LIN {X 0,Y 29.137,Z 512.707,A -85,B 0,C 180,E1 -30448.847,E2 -30448.847} C_VEL
LIN {X 0,Y 29.364,Z 512.686,A -85,B 0,C 180,E1 -30465.896,E2 -30465.896} C_VEL
LIN {X 0,Y 29.491,Z 512.673,A -85,B 0,C 180,E1 -30481.532,E2 -30481.532} C_VEL
LIN {X 0,Y 29.866,Z 512.638,A -85,B 0,C 180,E1 -30490.278,E2 -30490.278} C_VEL
LIN {X 0,Y 30.108,Z 512.614,A -85,B 0,C 180,E1 -30496.498,E2 -30496.498} C_VEL
LIN {X 0,Y 30.819,Z 512.551,A -85,B 0,C 180,E1 -30509.997,E2 -30509.997} C_VEL
LIN {X 0,Y 30.107,Z 512.614,A -85,B 0,C 180,E1 -30523.496,E2 -30523.496} C_VEL
LIN {X 0,Y 29.865,Z 512.638,A -85,B 0,C 180,E1 -30529.719,E2 -30529.719} C_VEL
LIN {X 0,Y 29.497,Z 512.672,A -85,B 0,C 180,E1 -30538.455,E2 -30538.455} C_VEL
LIN {X 0,Y 29.542,Z 512.668,A -85,B 0,C 180,E1 -30555.532,E2 -30555.532} C_VEL
LIN {X 0,Y 29.509,Z 512.672,A -85,B 0,C 180,E1 -30571.55,E2 -30571.55} C_VEL
LIN {X 0,Y 29.889,Z 512.637,A -85,B 0,C 180,E1 -30580.135,E2 -30580.135} C_VEL
LIN {X 0,Y 30.127,Z 512.613,A -85,B 0,C 180,E1 -30586.506,E2 -30586.506} C_VEL
LIN {X 0,Y 30.832,Z 512.546,A -85,B 0,C 180,E1 -30599.997,E2 -30599.997} C_VEL
LIN {X 0,Y 30.113,Z 512.615,A -85,B 0,C 180,E1 -30613.493,E2 -30613.493} C_VEL
LIN {X 0,Y 29.881,Z 512.634,A -85,B 0,C 180,E1 -30619.824,E2 -30619.824} C_VEL
LIN {X 0,Y 29.596,Z 512.661,A -85,B 0,C 180,E1 -30628.352,E2 -30628.352} C_VEL
LIN {X 0,Y 29.771,Z 512.646,A -85,B 0,C 180,E1 -30645.085,E2 -30645.085} C_VEL
LIN {X 0,Y 29.262,Z 512.695,A -85,B 0,C 180,E1 -30661.295,E2 -30661.295} C_VEL
LIN {X 0,Y 32.849,Z 512.354,A -85,B 0,C 180,E1 -30690.003,E2 -30690.003} C_VEL
LIN {X 0,Y 36.123,Z 511.976,A -85,B 0,C 180,E1 -30697.46,E2 -30697.46} C_VEL
LIN {X 0,Y 40.623,Z 525.984,A -85,B 0,C 180,E1 -30705.043,E2 -30705.043} C_VEL
LIN {X 0,Y 44.717,Z 535.436,A -85,B 0,C 180,E1 -30709.94,E2 -30709.94} C_VEL
LIN {X 0,Y 45.374,Z 537.398,A -85,B 0,C 180,E1 -30711.726,E2 -30711.726} C_VEL
LIN {X 0,Y 45.551,Z 539.426,A -85,B 0,C 180,E1 -30715.522,E2 -30715.522} C_VEL
LIN {X 0,Y 46.079,Z 543.284,A -85,B 0,C 180,E1 -30729.122,E2 -30729.122} C_VEL
LIN {X 0,Y 46.519,Z 544.027,A -85,B 0,C 180,E1 -30730.943,E2 -30730.943} C_VEL
LIN {X 0,Y 41.353,Z 535.78,A -85,B 0,C 180,E1 -30740.411,E2 -30740.411} C_VEL
LIN {X 0,Y 37.433,Z 526.306,A -85,B 0,C 180,E1 -30750.475,E2 -30750.475} C_VEL
LIN {X 0,Y 34.454,Z 515.149,A -85,B 0,C 180,E1 -30761.417,E2 -30761.417} C_VEL
LIN {X 0,Y 33.229,Z 512.321,A -85,B 0,C 180,E1 -30762.501,E2 -30762.501} C_VEL
LIN {X 0,Y 28.493,Z 512.766,A -85,B 0,C 180,E1 -30770.64,E2 -30770.64} C_VEL
LIN {X 0,Y 22.399,Z 513.078,A -85,B 0,C 180,E1 -30799.715,E2 -30799.715} C_VEL
LIN {X 0,Y 21.954,Z 513.092,A -85,B 0,C 180,E1 -30819.817,E2 -30819.817} C_VEL
LIN {X 0,Y 22.082,Z 513.088,A -85,B 0,C 180,E1 -30830.46,E2 -30830.46} C_VEL
LIN {X 0,Y 22.813,Z 513.065,A -85,B 0,C 180,E1 -30852.053,E2 -30852.053} C_VEL
LIN {X 0,Y 23.588,Z 513.042,A -85,B 0,C 180,E1 -30869.996,E2 -30869.996} C_VEL
LIN {X 0,Y 22.813,Z 513.065,A -85,B 0,C 180,E1 -30887.939,E2 -30887.939} C_VEL
LIN {X 0,Y 22.195,Z 513.084,A -85,B 0,C 180,E1 -30909.288,E2 -30909.288} C_VEL
LIN {X 0,Y 22.198,Z 513.084,A -85,B 0,C 180,E1 -30920.708,E2 -30920.708} C_VEL
LIN {X 0,Y 22.841,Z 513.064,A -85,B 0,C 180,E1 -30942.075,E2 -30942.075} C_VEL
LIN {X 0,Y 23.599,Z 513.041,A -85,B 0,C 180,E1 -30959.996,E2 -30959.996} C_VEL
LIN {X 0,Y 22.832,Z 513.064,A -85,B 0,C 180,E1 -30977.923,E2 -30977.923} C_VEL
LIN {X 0,Y 22.35,Z 513.08,A -85,B 0,C 180,E1 -30998.963,E2 -30998.963} C_VEL
LIN {X 0,Y 22.198,Z 513.084,A -85,B 0,C 180,E1 -31010.718,E2 -31010.718} C_VEL
LIN {X 0,Y 22.403,Z 513.078,A -85,B 0,C 180,E1 -31031.721,E2 -31031.721} C_VEL
LIN {X 0,Y 28.705,Z 512.746,A -85,B 0,C 180,E1 -31061.685,E2 -31061.685} C_VEL
LIN {X 0,Y 32.285,Z 512.408,A -85,B 0,C 180,E1 -31067.624,E2 -31067.624} C_VEL
LIN {X 0,Y 37.981,Z 527.127,A -85,B 0,C 180,E1 -31074.946,E2 -31074.946} C_VEL
LIN {X 0,Y 41.96,Z 535.075,A -85,B 0,C 180,E1 -31078.652,E2 -31078.652} C_VEL
LIN {X 0,Y 44.765,Z 540.723,A -85,B 0,C 180,E1 -31084.008,E2 -31084.008} C_VEL
LIN {X 0,Y 46.079,Z 543.284,A -85,B 0,C 180,E1 -31089.122,E2 -31089.122} C_VEL
LIN {X 0,Y 46.089,Z 543.42,A -85,B 0,C 180,E1 -31091.075,E2 -31091.075} C_VEL
LIN {X 0,Y 45.247,Z 542.248,A -85,B 0,C 180,E1 -31094.065,E2 -31094.065} C_VEL
LIN {X 0,Y 43.199,Z 539.068,A -85,B 0,C 180,E1 -31097.373,E2 -31097.373} C_VEL
LIN {X 0,Y 41.505,Z 536.26,A -85,B 0,C 180,E1 -31098.941,E2 -31098.941} C_VEL
LIN {X 0,Y 36.276,Z 526.902,A -85,B 0,C 180,E1 -31101.775,E2 -31101.775} C_VEL
LIN {X 0,Y 32.939,Z 519.69,A -85,B 0,C 180,E1 -31105.284,E2 -31105.284} C_VEL
LIN {X 0,Y 32.098,Z 517.339,A -85,B 0,C 180,E1 -31107.281,E2 -31107.281} C_VEL
LIN {X 0,Y 31.098,Z 514.138,A -85,B 0,C 180,E1 -31110.375,E2 -31110.375} C_VEL
LIN {X 0,Y 30.237,Z 512.601,A -85,B 0,C 180,E1 -31110.883,E2 -31110.883} C_VEL
LIN {X 0,Y 22.116,Z 513.086,A -85,B 0,C 180,E1 -31122.443,E2 -31122.443} C_VEL
LIN {X 0,Y 14.771,Z 513.178,A -85,B 0,C 180,E1 -31168.419,E2 -31168.419} C_VEL
LIN {X 0,Y 15.022,Z 513.178,A -85,B 0,C 180,E1 -31202.098,E2 -31202.098} C_VEL
LIN {X 0,Y 15.244,Z 513.178,A -85,B 0,C 180,E1 -31207.249,E2 -31207.249} C_VEL
LIN {X 0,Y 16.257,Z 513.178,A -85,B 0,C 180,E1 -31229.995,E2 -31229.995} C_VEL
LIN {X 0,Y 15.259,Z 513.178,A -85,B 0,C 180,E1 -31252.883,E2 -31252.883} C_VEL
LIN {X 0,Y 15.069,Z 513.178,A -85,B 0,C 180,E1 -31257.793,E2 -31257.793} C_VEL
LIN {X 0,Y 15.109,Z 513.178,A -85,B 0,C 180,E1 -31292.272,E2 -31292.272} C_VEL
LIN {X 0,Y 15.287,Z 513.178,A -85,B 0,C 180,E1 -31296.832,E2 -31296.832} C_VEL
LIN {X 0,Y 16.27,Z 513.178,A -85,B 0,C 180,E1 -31319.994,E2 -31319.994} C_VEL
LIN {X 0,Y 15.327,Z 513.178,A -85,B 0,C 180,E1 -31343.512,E2 -31343.512} C_VEL
LIN {X 0,Y 15.193,Z 513.178,A -85,B 0,C 180,E1 -31347.547,E2 -31347.547} C_VEL
LIN {X 0,Y 14.854,Z 513.178,A -85,B 0,C 180,E1 -31381.769,E2 -31381.769} C_VEL
LIN {X 0,Y 22.46,Z 513.076,A -85,B 0,C 180,E1 -31430.174,E2 -31430.174} C_VEL
LIN {X 0,Y 29.81,Z 512.644,A -85,B 0,C 180,E1 -31440.083,E2 -31440.083} C_VEL
LIN {X 0,Y 36.206,Z 526.908,A -85,B 0,C 180,E1 -31445.618,E2 -31445.618} C_VEL
LIN {X 0,Y 39.328,Z 532.669,A -85,B 0,C 180,E1 -31447.614,E2 -31447.614} C_VEL
LIN {X 0,Y 40.183,Z 534.194,A -85,B 0,C 180,E1 -31448.555,E2 -31448.555} C_VEL
LIN {X 0,Y 39.303,Z 532.936,A -85,B 0,C 180,E1 -31451.585,E2 -31451.585} C_VEL
LIN {X 0,Y 35.167,Z 525.313,A -85,B 0,C 180,E1 -31459.499,E2 -31459.499} C_VEL
LIN {X 0,Y 32.098,Z 517.339,A -85,B 0,C 180,E1 -31467.281,E2 -31467.281} C_VEL
LIN {X 0,Y 30.488,Z 515.25,A -85,B 0,C 180,E1 -31469.778,E2 -31469.778} C_VEL
LIN {X 0,Y 27.216,Z 513.761,A -85,B 0,C 180,E1 -31473.03,E2 -31473.03} C_VEL
LIN {X 0,Y 21.887,Z 513.154,A -85,B 0,C 180,E1 -31477.951,E2 -31477.951} C_VEL
LIN {X 0,Y 8.626,Z 513.183,A -85,B 0,C 180,E1 -31512.093,E2 -31512.093} C_VEL
LIN {X 0,Y 7.17,Z 513.178,A -85,B 0,C 180,E1 -31543.705,E2 -31543.705} C_VEL
LIN {X 0,Y 7.725,Z 513.178,A -85,B 0,C 180,E1 -31565.507,E2 -31565.507} C_VEL
LIN {X 0,Y 8.68,Z 513.178,A -85,B 0,C 180,E1 -31589.99,E2 -31589.99} C_VEL
LIN {X 0,Y 7.768,Z 513.178,A -85,B 0,C 180,E1 -31615.182,E2 -31615.182} C_VEL
LIN {X 0,Y 7.778,Z 513.178,A -85,B 0,C 180,E1 -31654.607,E2 -31654.607} C_VEL
LIN {X 0,Y 8.704,Z 513.178,A -85,B 0,C 180,E1 -31679.989,E2 -31679.989} C_VEL
LIN {X 0,Y 7.787,Z 513.178,A -85,B 0,C 180,E1 -31705.527,E2 -31705.527} C_VEL
LIN {X 0,Y 7.689,Z 513.178,A -85,B 0,C 180,E1 -31746.031,E2 -31746.031} C_VEL
LIN {X 0,Y 21.814,Z 513.097,A -85,B 0,C 180,E1 -31810.123,E2 -31810.123} C_VEL
LIN {X 0,Y 29.056,Z 512.844,A -85,B 0,C 180,E1 -31813.979,E2 -31813.979} C_VEL
LIN {X 0,Y 30.01,Z 515.063,A -85,B 0,C 180,E1 -31814.637,E2 -31814.637} C_VEL
LIN {X 0,Y 30.002,Z 515.028,A -85,B 0,C 180,E1 -31815.529,E2 -31815.529} C_VEL
LIN {X 0,Y 28.961,Z 512.723,A -85,B 0,C 180,E1 -31817.295,E2 -31817.295} C_VEL
LIN {X 0,Y 22.359,Z 513.079,A -85,B 0,C 180,E1 -31821.055,E2 -31821.055} C_VEL
LIN {X 0,Y 7.651,Z 513.178,A -85,B 0,C 180,E1 -31883.252,E2 -31883.252} C_VEL
LIN {X 0,Y 7.17,Z 513.178,A -85,B 0,C 180,E1 -31903.705,E2 -31903.705} C_VEL
LIN {X 0,Y 6.425,Z 513.178,A -85,B 0,C 180,E1 -31914.755,E2 -31914.755} C_VEL
LIN {X 0,Y 3.928,Z 513.178,A -85,B 0,C 180,E1 -31933.058,E2 -31933.058} C_VEL
LIN {X 0,Y 1.474,Z 513.178,A -85,B 0,C 180,E1 -31968.947,E2 -31968.947} C_VEL
LIN {X 0,Y 0.256,Z 513.178,A -85,B 0,C 180,E1 -32039.624,E2 -32039.624} C_VEL
LIN {X 0,Y 0.23,Z 513.178,A -85,B 0,C 180,E1 -32130.384,E2 -32130.384} C_VEL
LIN {X 0,Y 0.139,Z 513.178,A -85,B 0,C 180,E1 -32309.367,E2 -32309.367} C_VEL
LIN {X 0,Y 0.256,Z 513.178,A -85,B 0,C 180,E1 -32399.624,E2 -32399.624} C_VEL
LIN {X 0,Y 2.228,Z 515.178,A -85,B 0,C 180,E1 -32424.946,E2 -32424.946} C_VEL
LIN {X 0,Y 2.228,Z 600,A -85,B 0,C 180,E1 -32424.946,E2 -32424.946} C_VEL
LIN {X 0,Y 2.228,Z 600,A -85,B 0,C 180,E1 -32424.946,E2 -32424.946}

QRS_NEXT_CUT()

QRS_NEXT()
QRS_HOME()

END
